// TwinCAT 3 PLC project p1
// ProgramVersion: 3.1.4023.0
// libraries:
//   Tc2_ControllerToolbox, * (Beckhoff Automation GmbH)
//   Tc2_EtherCAT, * (Beckhoff Automation GmbH)
//   Tc2_MC2, * (Beckhoff Automation GmbH)
//   Tc2_Standard, * (Beckhoff Automation GmbH)
//   Tc2_System, * (Beckhoff Automation GmbH)
//   Tc2_Utilities, * (Beckhoff Automation GmbH)
//   Tc3_Module, * (Beckhoff Automation GmbH)
// project tree:
//   DUTs/UR_10 _O2T_Registers/ UR_10_O2T_Registers.TcDUT, UR_O2T_bits_2.TcDUT, UR_O2T_floats_2.TcDUT, UR_O2T_int_2.TcDUT
//   DUTs/UR_3_T2O_Joints/ UR_3_T2O_Joints.TcDUT
//   DUTs/UR_4_T2O_TCP/ UR_4_T2O_TCP.TcDUT
//   DUTs/UR_5_T2O_BitRegisters/ UR_5_T2O_BitRegisters.TcDUT
//   DUTs/UR_6_T2O_IntRegisters/ UR_6_T2O_IntRegisters.TcDUT
//   DUTs/UR_7_T2O_FloatRegisters/ UR_7_T2O_FloatRegisters.TcDUT
//   DUTs/UR_9_O2T_Registers/ UR_9_O2T_Registers.TcDUT, UR_O2T_bits.TcDUT, UR_O2T_floats.TcDUT, UR_O2T_int.TcDUT
//   DUTs/Vision Struct/ ck_real_flag_data.TcDUT, Vision_data.TcDUT, Vision_flags.TcDUT, Vision_int_state.TcDUT
//   GVLs/MainProg Params/Constans/ VFUNCTION.TcGVL, _FUNCTION.TcGVL
//   GVLs/MainProg Params/Variables/ GLV_USER_FUN.TcGVL
//   GVLs/miscellaneus/ data_to_robot.TcGVL, Global_actual_velocity.TcGVL
//   GVLs/QRob/ QrCts.TcGVL
//   GVLs/QRob/Variables/ Global_Servo.TcGVL, QrRetVarState.TcGVL
//   GVLs/Robot Params/Constans/ RCts.TcGVL
//   GVLs/Robot Params/Variables/ Robot_UR5.TcGVL, Robot_UR3.TcGVL, UR3RetVarState.TcGVL, UR5RetVarState.TcGVL (not stored)
//   GVLs/Vision Params/Constants/ VCts.TcGVL
//   GVLs/Vision Params/Structs/ Vision_struct.TcGVL
//   GVLs/Vision Params/Variables/ VisionRetVarState.TcGVL
//   / PlcTask.TcTTO
//   POUs/POUs/Fuzzy/ Subsystem.TcPOU, trimf.TcPOU, trimf_l.TcPOU
//   POUs/POUs/IR_take_img/ get_images.TcPOU
//   POUs/POUs/l/ Atornillar_ur5.TcPOU, data_robot_ur5.TcPOU, data_robot_ur3.TcPOU, flip_byte_int.TcPOU, flip_real.TcPOU, flip_byte.TcPOU, flip_int.TcPOU, pulse_.TcPOU, limit_current.TcPOU
//   POUs/POUs/ MASTER_CTR.TcPOU
//   POUs/POUs/miscellaneous/ POU.TcPOU, profinet_UR3.TcPOU, profinet_UR5.TcPOU, UR3_Robot.TcPOU, UR5_robot.TcPOU
//   POUs/POUs/Qrob/QRob_functions/ Get_QRob_Pos.TcPOU, Temperature_Ctr.TcPOU, Qrob_control.TcPOU
//   POUs/POUs/Qrob/Qrob_State_Machine/ QRob_StateMachine.TcPOU
//   POUs/POUs/ROBOTS/Robot_functions/ ck_state.TcPOU, read_bool_flag.TcPOU, read_bool_flag_move.TcPOU, write_bool_flag.TcPOU, wr_GL_STATE.TcPOU (not stored), wr_state.TcPOU
//   POUs/POUs/ROBOTS/Robot_machine_state/ UR3_StateMachine.TcPOU, UR5_StateMachine.TcPOU
//   POUs/POUs/VISION/Vision_functions/ ck_state_v.TcPOU, ck_real_value.TcPOU, wr_real_value.TcPOU, wr_state_v.TcPOU
//   POUs/POUs/VISION/Vision_machines_states/ Vision_StateMachine.TcPOU
// real-time tasks:
//   TASK PlcTask2: cycle T#1ms, priority 4, ADS port 352
// motion (NC):
//   TASK NC-Task 1 SAF: cycle T#2ms, priority 6, ADS port 501
//   TASK NC-Task 1 SVB: cycle T#10ms, priority 10, ADS port 511
//   AXIS Axis 1 (id 1)
//     General: UnitName=°
//     Dynamic: Acceleration=321.75, Deceleration=321.75, Jerk=1070.01, FastAxisStopSignalType=3
//     Velo: RefSearch=70, RefSync=120, Fast=200, Maximum=225
//     PositionAreaControl: Enable=false
//     TargetPosControl: Enable=false
//     OtherSettings: AllowMotionCmdToSlave=true, DataPersistence=true
//     encoder EncType=19
//       EncPara: ScaleFactorNumerator=0.000686648, MaxCount=#xffffffff, ReferenceSystem=4
//         Inc: RefSyncInverse=false
//     drive DrvType=16
//       DrvPara: MaxCount=#xffffffff, DriveControlDWord=#x00020000
//         Analog: VeloReferenz=225, TorqueSetpointScale=1, ScaleFactorActTorque=1
//         TimeComp: TaskDelayCycles=1
//     controller CtrType=1
//       CtrPara: PriorControlFactor=1
//         PosDiffControl: Enable=false
//         Observer: BandWidth=20
// I/O:
//   DEVICE Device 5 (EtherCAT), AmsNetId 172.18.236.0.6.1
//     Drive 1 (ZeroErr Driver) [ZeroErr Driver]
//   DEVICE Device 7 (EtherCAT), AmsNetId 172.18.236.0.8.1
//     Term 4 (EK1100) [EK1100 EtherCAT Coupler (2A E-Bus)]
//       Term 5 (EL2809) [EL2809 16Ch. Dig. Output 24V, 0.5A]
//       Term 12 (EL1809) [EL1809 16Ch. Dig. Input 24V, 3ms]
//       Term 6 (EL6001) [EL6001 Interface (RS232)]
//       Term 4 (EL6631) [EL6631 PROFINET IO Controller]
//       Term 5 (EL6751) [EL6751 CANopen Master]
//       Term 6 (EL9011) [EL9011 End Terminal]
//   DEVICE Device 4 (EL6631), AmsNetId 172.18.236.0.5.1
//     uriodev1ur5 [Universal Robots A/S UR IO device, for PNIO controller with PDev 00000]
//       modules: Term 1 (DAP Module), Term 3 (1_T2O State), Term 4 (2_T2O IO), Term 5 (3_T2O Joints), Term 6 (4_T2O TCP), Term 7 (5_T2O General Purpose Bit Registers), Term 8 (6_T2O General Purpose Int Registers), Term 9 (7_T2O General Purpose Float Registers), Term 10 (8_O2T Robot IO), Term 11 (9_O2T General Purpose Registers 1), Term 12 (10_O2T General Purpose Registers 2)
//     uriodev1ur3 [Universal Robots A/S UR IO device, for PNIO controller with PDev 00000]
//       modules: Term 2 (DAP Module), Term 13 (1_T2O State), Term 14 (2_T2O IO), Term 15 (3_T2O Joints), Term 16 (4_T2O TCP), Term 17 (5_T2O General Purpose Bit Registers), Term 18 (6_T2O General Purpose Int Registers), Term 19 (7_T2O General Purpose Float Registers), Term 20 (8_O2T Robot IO), Term 21 (9_O2T General Purpose Registers 1), Term 22 (10_O2T General Purpose Registers 2)
// variable links:
//   NC-Task 1 SAF/Axes/Axis 1 <-> Device 5 (EtherCAT)/Drive 1 (ZeroErr Driver)
//     Drive/Inputs/In/nDataIn3[0] <-> Transmit PDO mapping 0/Torque Actual Value
//     Drive/Inputs/In/nDcOutputTime <-> InfoData/DcOutputShift
//     Drive/Inputs/In/nState1 <-> Transmit PDO mapping 0/Status word
//     Drive/Inputs/In/nState2 <-> Transmit PDO mapping 0/Status word @bit 8
//     Drive/Inputs/In/nState4 @bit 1 <-> WcState/InputToggle
//     Drive/Inputs/In/nState4 <-> WcState/WcState
//     Drive/Inputs/In/nState5 <-> Transmit PDO mapping 0/Modes of operation display
//     Drive/Outputs/Out/nCtrl1 <-> Receive PDO mapping 0/Control word
//     Drive/Outputs/Out/nCtrl2 <-> Receive PDO mapping 0/Control word @bit 8
//     Drive/Outputs/Out/nCtrl5 <-> Receive PDO mapping 0/Modes of operation
//     Drive/Outputs/Out/nDataOut1 <-> Receive PDO mapping 0/Target Position
//     Drive/Outputs/Out/nDataOut3[0] <-> Receive PDO mapping 0/Torque Offset
//     Drive/Outputs/Out/nDataOut4[0] <-> Receive PDO mapping 0/Target Torque
//     Enc/Inputs/In/nDataIn1 <-> Transmit PDO mapping 0/Position actual value
//     Enc/Inputs/In/nDataIn7 <-> Transmit PDO mapping 0/Actual velocity
//     Enc/Inputs/In/nDcInputTime <-> InfoData/DcInputShift
//     Enc/Inputs/In/nState4 @bit 1 <-> WcState/InputToggle
//     Enc/Inputs/In/nState4 <-> WcState/WcState
//   p1/p1 Instance <-> Device 4 (EL6631)/uriodev1ur3
//     PlcTask Inputs/Robot_UR3.UR_TCP/FLOAT14[0] <-> API/Term 16 (4_T2O TCP)/Subterm 20 (4_T2O TCP)/Inputs/T2O TCP[56]
//     PlcTask Inputs/Robot_UR3.UR_TCP/FLOAT14[1] <-> API/Term 16 (4_T2O TCP)/Subterm 20 (4_T2O TCP)/Inputs/T2O TCP[57]
//     PlcTask Inputs/Robot_UR3.UR_TCP/FLOAT14[2] <-> API/Term 16 (4_T2O TCP)/Subterm 20 (4_T2O TCP)/Inputs/T2O TCP[58]
//     PlcTask Inputs/Robot_UR3.UR_TCP/FLOAT14[3] <-> API/Term 16 (4_T2O TCP)/Subterm 20 (4_T2O TCP)/Inputs/T2O TCP[59]
//     PlcTask Inputs/Robot_UR3.UR_TCP/FLOAT15[0] <-> API/Term 16 (4_T2O TCP)/Subterm 20 (4_T2O TCP)/Inputs/T2O TCP[60]
//     PlcTask Inputs/Robot_UR3.UR_TCP/FLOAT15[1] <-> API/Term 16 (4_T2O TCP)/Subterm 20 (4_T2O TCP)/Inputs/T2O TCP[61]
//     PlcTask Inputs/Robot_UR3.UR_TCP/FLOAT15[2] <-> API/Term 16 (4_T2O TCP)/Subterm 20 (4_T2O TCP)/Inputs/T2O TCP[62]
//     PlcTask Inputs/Robot_UR3.UR_TCP/FLOAT15[3] <-> API/Term 16 (4_T2O TCP)/Subterm 20 (4_T2O TCP)/Inputs/T2O TCP[63]
//     PlcTask Inputs/Robot_UR3.UR_TCP/FLOAT16[0] <-> API/Term 16 (4_T2O TCP)/Subterm 20 (4_T2O TCP)/Inputs/T2O TCP[64]
//     PlcTask Inputs/Robot_UR3.UR_TCP/FLOAT16[1] <-> API/Term 16 (4_T2O TCP)/Subterm 20 (4_T2O TCP)/Inputs/T2O TCP[65]
//     PlcTask Inputs/Robot_UR3.UR_TCP/FLOAT16[2] <-> API/Term 16 (4_T2O TCP)/Subterm 20 (4_T2O TCP)/Inputs/T2O TCP[66]
//     PlcTask Inputs/Robot_UR3.UR_TCP/FLOAT16[3] <-> API/Term 16 (4_T2O TCP)/Subterm 20 (4_T2O TCP)/Inputs/T2O TCP[67]
//     PlcTask Inputs/Robot_UR3.UR_TCP/FLOAT17[0] <-> API/Term 16 (4_T2O TCP)/Subterm 20 (4_T2O TCP)/Inputs/T2O TCP[68]
//     PlcTask Inputs/Robot_UR3.UR_TCP/FLOAT17[1] <-> API/Term 16 (4_T2O TCP)/Subterm 20 (4_T2O TCP)/Inputs/T2O TCP[69]
//     PlcTask Inputs/Robot_UR3.UR_TCP/FLOAT17[2] <-> API/Term 16 (4_T2O TCP)/Subterm 20 (4_T2O TCP)/Inputs/T2O TCP[70]
//     PlcTask Inputs/Robot_UR3.UR_TCP/FLOAT17[3] <-> API/Term 16 (4_T2O TCP)/Subterm 20 (4_T2O TCP)/Inputs/T2O TCP[71]
//     PlcTask Inputs/Robot_UR3.UR_TCP/FLOAT18[0] <-> API/Term 16 (4_T2O TCP)/Subterm 20 (4_T2O TCP)/Inputs/T2O TCP[72]
//     PlcTask Inputs/Robot_UR3.UR_TCP/FLOAT18[1] <-> API/Term 16 (4_T2O TCP)/Subterm 20 (4_T2O TCP)/Inputs/T2O TCP[73]
//     PlcTask Inputs/Robot_UR3.UR_TCP/FLOAT18[2] <-> API/Term 16 (4_T2O TCP)/Subterm 20 (4_T2O TCP)/Inputs/T2O TCP[74]
//     PlcTask Inputs/Robot_UR3.UR_TCP/FLOAT18[3] <-> API/Term 16 (4_T2O TCP)/Subterm 20 (4_T2O TCP)/Inputs/T2O TCP[75]
//     PlcTask Inputs/Robot_UR3.UR_outputs/B{0..56 step 8} <-> API/Term 17 (5_T2O General Purpose Bit Registers)/Subterm 21 (5_T2O General Purpose Bit Registers)/Inputs/T2O Bit Registers[{0..7}]  (8 links)
//     PlcTask Inputs/Robot_UR3.UR_outputs/B1 <-> API/Term 17 (5_T2O General Purpose Bit Registers)/Subterm 21 (5_T2O General Purpose Bit Registers)/Inputs/T2O Bit Registers[0] @bit 1
//     PlcTask Inputs/Robot_UR3.UR_outputs/B10 <-> API/Term 17 (5_T2O General Purpose Bit Registers)/Subterm 21 (5_T2O General Purpose Bit Registers)/Inputs/T2O Bit Registers[1] @bit 2
//     PlcTask Inputs/Robot_UR3.UR_outputs/B11 <-> API/Term 17 (5_T2O General Purpose Bit Registers)/Subterm 21 (5_T2O General Purpose Bit Registers)/Inputs/T2O Bit Registers[1] @bit 3
//     PlcTask Inputs/Robot_UR3.UR_outputs/B12 <-> API/Term 17 (5_T2O General Purpose Bit Registers)/Subterm 21 (5_T2O General Purpose Bit Registers)/Inputs/T2O Bit Registers[1] @bit 4
//     PlcTask Inputs/Robot_UR3.UR_outputs/B13 <-> API/Term 17 (5_T2O General Purpose Bit Registers)/Subterm 21 (5_T2O General Purpose Bit Registers)/Inputs/T2O Bit Registers[1] @bit 5
//     PlcTask Inputs/Robot_UR3.UR_outputs/B14 <-> API/Term 17 (5_T2O General Purpose Bit Registers)/Subterm 21 (5_T2O General Purpose Bit Registers)/Inputs/T2O Bit Registers[1] @bit 6
//     PlcTask Inputs/Robot_UR3.UR_outputs/B15 <-> API/Term 17 (5_T2O General Purpose Bit Registers)/Subterm 21 (5_T2O General Purpose Bit Registers)/Inputs/T2O Bit Registers[1] @bit 7
//     PlcTask Inputs/Robot_UR3.UR_outputs/B17 <-> API/Term 17 (5_T2O General Purpose Bit Registers)/Subterm 21 (5_T2O General Purpose Bit Registers)/Inputs/T2O Bit Registers[2] @bit 1
//     PlcTask Inputs/Robot_UR3.UR_outputs/B18 <-> API/Term 17 (5_T2O General Purpose Bit Registers)/Subterm 21 (5_T2O General Purpose Bit Registers)/Inputs/T2O Bit Registers[2] @bit 2
//     PlcTask Inputs/Robot_UR3.UR_outputs/B19 <-> API/Term 17 (5_T2O General Purpose Bit Registers)/Subterm 21 (5_T2O General Purpose Bit Registers)/Inputs/T2O Bit Registers[2] @bit 3
//     PlcTask Inputs/Robot_UR3.UR_outputs/B2 <-> API/Term 17 (5_T2O General Purpose Bit Registers)/Subterm 21 (5_T2O General Purpose Bit Registers)/Inputs/T2O Bit Registers[0] @bit 2
//     PlcTask Inputs/Robot_UR3.UR_outputs/B20 <-> API/Term 17 (5_T2O General Purpose Bit Registers)/Subterm 21 (5_T2O General Purpose Bit Registers)/Inputs/T2O Bit Registers[2] @bit 4
//     PlcTask Inputs/Robot_UR3.UR_outputs/B21 <-> API/Term 17 (5_T2O General Purpose Bit Registers)/Subterm 21 (5_T2O General Purpose Bit Registers)/Inputs/T2O Bit Registers[2] @bit 5
//     PlcTask Inputs/Robot_UR3.UR_outputs/B22 <-> API/Term 17 (5_T2O General Purpose Bit Registers)/Subterm 21 (5_T2O General Purpose Bit Registers)/Inputs/T2O Bit Registers[2] @bit 6
//     PlcTask Inputs/Robot_UR3.UR_outputs/B23 <-> API/Term 17 (5_T2O General Purpose Bit Registers)/Subterm 21 (5_T2O General Purpose Bit Registers)/Inputs/T2O Bit Registers[2] @bit 7
//     PlcTask Inputs/Robot_UR3.UR_outputs/B25 <-> API/Term 17 (5_T2O General Purpose Bit Registers)/Subterm 21 (5_T2O General Purpose Bit Registers)/Inputs/T2O Bit Registers[3] @bit 1
//     PlcTask Inputs/Robot_UR3.UR_outputs/B26 <-> API/Term 17 (5_T2O General Purpose Bit Registers)/Subterm 21 (5_T2O General Purpose Bit Registers)/Inputs/T2O Bit Registers[3] @bit 2
//     PlcTask Inputs/Robot_UR3.UR_outputs/B27 <-> API/Term 17 (5_T2O General Purpose Bit Registers)/Subterm 21 (5_T2O General Purpose Bit Registers)/Inputs/T2O Bit Registers[3] @bit 3
//     PlcTask Inputs/Robot_UR3.UR_outputs/B28 <-> API/Term 17 (5_T2O General Purpose Bit Registers)/Subterm 21 (5_T2O General Purpose Bit Registers)/Inputs/T2O Bit Registers[3] @bit 4
//     PlcTask Inputs/Robot_UR3.UR_outputs/B29 <-> API/Term 17 (5_T2O General Purpose Bit Registers)/Subterm 21 (5_T2O General Purpose Bit Registers)/Inputs/T2O Bit Registers[3] @bit 5
//     PlcTask Inputs/Robot_UR3.UR_outputs/B3 <-> API/Term 17 (5_T2O General Purpose Bit Registers)/Subterm 21 (5_T2O General Purpose Bit Registers)/Inputs/T2O Bit Registers[0] @bit 3
//     PlcTask Inputs/Robot_UR3.UR_outputs/B30 <-> API/Term 17 (5_T2O General Purpose Bit Registers)/Subterm 21 (5_T2O General Purpose Bit Registers)/Inputs/T2O Bit Registers[3] @bit 6
//     PlcTask Inputs/Robot_UR3.UR_outputs/B31 <-> API/Term 17 (5_T2O General Purpose Bit Registers)/Subterm 21 (5_T2O General Purpose Bit Registers)/Inputs/T2O Bit Registers[3] @bit 7
//     PlcTask Inputs/Robot_UR3.UR_outputs/B33 <-> API/Term 17 (5_T2O General Purpose Bit Registers)/Subterm 21 (5_T2O General Purpose Bit Registers)/Inputs/T2O Bit Registers[4] @bit 1
//     PlcTask Inputs/Robot_UR3.UR_outputs/B34 <-> API/Term 17 (5_T2O General Purpose Bit Registers)/Subterm 21 (5_T2O General Purpose Bit Registers)/Inputs/T2O Bit Registers[4] @bit 2
//     PlcTask Inputs/Robot_UR3.UR_outputs/B35 <-> API/Term 17 (5_T2O General Purpose Bit Registers)/Subterm 21 (5_T2O General Purpose Bit Registers)/Inputs/T2O Bit Registers[4] @bit 3
//     PlcTask Inputs/Robot_UR3.UR_outputs/B36 <-> API/Term 17 (5_T2O General Purpose Bit Registers)/Subterm 21 (5_T2O General Purpose Bit Registers)/Inputs/T2O Bit Registers[4] @bit 4
//     PlcTask Inputs/Robot_UR3.UR_outputs/B37 <-> API/Term 17 (5_T2O General Purpose Bit Registers)/Subterm 21 (5_T2O General Purpose Bit Registers)/Inputs/T2O Bit Registers[4] @bit 5
//     PlcTask Inputs/Robot_UR3.UR_outputs/B38 <-> API/Term 17 (5_T2O General Purpose Bit Registers)/Subterm 21 (5_T2O General Purpose Bit Registers)/Inputs/T2O Bit Registers[4] @bit 6
//     PlcTask Inputs/Robot_UR3.UR_outputs/B39 <-> API/Term 17 (5_T2O General Purpose Bit Registers)/Subterm 21 (5_T2O General Purpose Bit Registers)/Inputs/T2O Bit Registers[4] @bit 7
//     PlcTask Inputs/Robot_UR3.UR_outputs/B4 <-> API/Term 17 (5_T2O General Purpose Bit Registers)/Subterm 21 (5_T2O General Purpose Bit Registers)/Inputs/T2O Bit Registers[0] @bit 4
//     PlcTask Inputs/Robot_UR3.UR_outputs/B41 <-> API/Term 17 (5_T2O General Purpose Bit Registers)/Subterm 21 (5_T2O General Purpose Bit Registers)/Inputs/T2O Bit Registers[5] @bit 1
//     PlcTask Inputs/Robot_UR3.UR_outputs/B42 <-> API/Term 17 (5_T2O General Purpose Bit Registers)/Subterm 21 (5_T2O General Purpose Bit Registers)/Inputs/T2O Bit Registers[5] @bit 2
//     PlcTask Inputs/Robot_UR3.UR_outputs/B43 <-> API/Term 17 (5_T2O General Purpose Bit Registers)/Subterm 21 (5_T2O General Purpose Bit Registers)/Inputs/T2O Bit Registers[5] @bit 3
//     PlcTask Inputs/Robot_UR3.UR_outputs/B44 <-> API/Term 17 (5_T2O General Purpose Bit Registers)/Subterm 21 (5_T2O General Purpose Bit Registers)/Inputs/T2O Bit Registers[5] @bit 4
//     PlcTask Inputs/Robot_UR3.UR_outputs/B45 <-> API/Term 17 (5_T2O General Purpose Bit Registers)/Subterm 21 (5_T2O General Purpose Bit Registers)/Inputs/T2O Bit Registers[5] @bit 5
//     PlcTask Inputs/Robot_UR3.UR_outputs/B46 <-> API/Term 17 (5_T2O General Purpose Bit Registers)/Subterm 21 (5_T2O General Purpose Bit Registers)/Inputs/T2O Bit Registers[5] @bit 6
//     PlcTask Inputs/Robot_UR3.UR_outputs/B47 <-> API/Term 17 (5_T2O General Purpose Bit Registers)/Subterm 21 (5_T2O General Purpose Bit Registers)/Inputs/T2O Bit Registers[5] @bit 7
//     PlcTask Inputs/Robot_UR3.UR_outputs/B49 <-> API/Term 17 (5_T2O General Purpose Bit Registers)/Subterm 21 (5_T2O General Purpose Bit Registers)/Inputs/T2O Bit Registers[6] @bit 1
//     PlcTask Inputs/Robot_UR3.UR_outputs/B5 <-> API/Term 17 (5_T2O General Purpose Bit Registers)/Subterm 21 (5_T2O General Purpose Bit Registers)/Inputs/T2O Bit Registers[0] @bit 5
//     PlcTask Inputs/Robot_UR3.UR_outputs/B50 <-> API/Term 17 (5_T2O General Purpose Bit Registers)/Subterm 21 (5_T2O General Purpose Bit Registers)/Inputs/T2O Bit Registers[6] @bit 2
//     PlcTask Inputs/Robot_UR3.UR_outputs/B51 <-> API/Term 17 (5_T2O General Purpose Bit Registers)/Subterm 21 (5_T2O General Purpose Bit Registers)/Inputs/T2O Bit Registers[6] @bit 3
//     PlcTask Inputs/Robot_UR3.UR_outputs/B52 <-> API/Term 17 (5_T2O General Purpose Bit Registers)/Subterm 21 (5_T2O General Purpose Bit Registers)/Inputs/T2O Bit Registers[6] @bit 4
//     PlcTask Inputs/Robot_UR3.UR_outputs/B53 <-> API/Term 17 (5_T2O General Purpose Bit Registers)/Subterm 21 (5_T2O General Purpose Bit Registers)/Inputs/T2O Bit Registers[6] @bit 5
//     PlcTask Inputs/Robot_UR3.UR_outputs/B54 <-> API/Term 17 (5_T2O General Purpose Bit Registers)/Subterm 21 (5_T2O General Purpose Bit Registers)/Inputs/T2O Bit Registers[6] @bit 6
//     PlcTask Inputs/Robot_UR3.UR_outputs/B55 <-> API/Term 17 (5_T2O General Purpose Bit Registers)/Subterm 21 (5_T2O General Purpose Bit Registers)/Inputs/T2O Bit Registers[6] @bit 7
//     PlcTask Inputs/Robot_UR3.UR_outputs/B57 <-> API/Term 17 (5_T2O General Purpose Bit Registers)/Subterm 21 (5_T2O General Purpose Bit Registers)/Inputs/T2O Bit Registers[7] @bit 1
//     PlcTask Inputs/Robot_UR3.UR_outputs/B58 <-> API/Term 17 (5_T2O General Purpose Bit Registers)/Subterm 21 (5_T2O General Purpose Bit Registers)/Inputs/T2O Bit Registers[7] @bit 2
//     PlcTask Inputs/Robot_UR3.UR_outputs/B59 <-> API/Term 17 (5_T2O General Purpose Bit Registers)/Subterm 21 (5_T2O General Purpose Bit Registers)/Inputs/T2O Bit Registers[7] @bit 3
//     PlcTask Inputs/Robot_UR3.UR_outputs/B6 <-> API/Term 17 (5_T2O General Purpose Bit Registers)/Subterm 21 (5_T2O General Purpose Bit Registers)/Inputs/T2O Bit Registers[0] @bit 6
//     PlcTask Inputs/Robot_UR3.UR_outputs/B60 <-> API/Term 17 (5_T2O General Purpose Bit Registers)/Subterm 21 (5_T2O General Purpose Bit Registers)/Inputs/T2O Bit Registers[7] @bit 4
//     PlcTask Inputs/Robot_UR3.UR_outputs/B61 <-> API/Term 17 (5_T2O General Purpose Bit Registers)/Subterm 21 (5_T2O General Purpose Bit Registers)/Inputs/T2O Bit Registers[7] @bit 5
//     PlcTask Inputs/Robot_UR3.UR_outputs/B62 <-> API/Term 17 (5_T2O General Purpose Bit Registers)/Subterm 21 (5_T2O General Purpose Bit Registers)/Inputs/T2O Bit Registers[7] @bit 6
//     PlcTask Inputs/Robot_UR3.UR_outputs/B63 <-> API/Term 17 (5_T2O General Purpose Bit Registers)/Subterm 21 (5_T2O General Purpose Bit Registers)/Inputs/T2O Bit Registers[7] @bit 7
//     PlcTask Inputs/Robot_UR3.UR_outputs/B7 <-> API/Term 17 (5_T2O General Purpose Bit Registers)/Subterm 21 (5_T2O General Purpose Bit Registers)/Inputs/T2O Bit Registers[0] @bit 7
//     PlcTask Inputs/Robot_UR3.UR_outputs/B9 <-> API/Term 17 (5_T2O General Purpose Bit Registers)/Subterm 21 (5_T2O General Purpose Bit Registers)/Inputs/T2O Bit Registers[1] @bit 1
//     PlcTask Inputs/Robot_UR3.UR_outputs_int/INT0[0] <-> API/Term 18 (6_T2O General Purpose Int Registers)/Subterm 22 (6_T2O General Purpose Int Registers)/Inputs/T2O Int Registers[0]
//     PlcTask Inputs/Robot_UR3.UR_outputs_int/INT0[1] <-> API/Term 18 (6_T2O General Purpose Int Registers)/Subterm 22 (6_T2O General Purpose Int Registers)/Inputs/T2O Int Registers[1]
//     PlcTask Inputs/Robot_UR3.UR_outputs_int/INT0[2] <-> API/Term 18 (6_T2O General Purpose Int Registers)/Subterm 22 (6_T2O General Purpose Int Registers)/Inputs/T2O Int Registers[2]
//     PlcTask Inputs/Robot_UR3.UR_outputs_int/INT0[3] <-> API/Term 18 (6_T2O General Purpose Int Registers)/Subterm 22 (6_T2O General Purpose Int Registers)/Inputs/T2O Int Registers[3]
//     PlcTask Inputs/Robot_UR3.UR_outputs_int/INT1[0] <-> API/Term 18 (6_T2O General Purpose Int Registers)/Subterm 22 (6_T2O General Purpose Int Registers)/Inputs/T2O Int Registers[4]
//     PlcTask Inputs/Robot_UR3.UR_outputs_int/INT1[1] <-> API/Term 18 (6_T2O General Purpose Int Registers)/Subterm 22 (6_T2O General Purpose Int Registers)/Inputs/T2O Int Registers[5]
//     PlcTask Inputs/Robot_UR3.UR_outputs_int/INT1[2] <-> API/Term 18 (6_T2O General Purpose Int Registers)/Subterm 22 (6_T2O General Purpose Int Registers)/Inputs/T2O Int Registers[6]
//     PlcTask Inputs/Robot_UR3.UR_outputs_int/INT1[3] <-> API/Term 18 (6_T2O General Purpose Int Registers)/Subterm 22 (6_T2O General Purpose Int Registers)/Inputs/T2O Int Registers[7]
//     PlcTask Inputs/Robot_UR3.UR_outputs_int/INT2[0] <-> API/Term 18 (6_T2O General Purpose Int Registers)/Subterm 22 (6_T2O General Purpose Int Registers)/Inputs/T2O Int Registers[8]
//     PlcTask Inputs/Robot_UR3.UR_outputs_int/INT2[1] <-> API/Term 18 (6_T2O General Purpose Int Registers)/Subterm 22 (6_T2O General Purpose Int Registers)/Inputs/T2O Int Registers[9]
//     PlcTask Inputs/Robot_UR3.UR_outputs_int/INT2[2] <-> API/Term 18 (6_T2O General Purpose Int Registers)/Subterm 22 (6_T2O General Purpose Int Registers)/Inputs/T2O Int Registers[10]
//     PlcTask Inputs/Robot_UR3.UR_outputs_int/INT2[3] <-> API/Term 18 (6_T2O General Purpose Int Registers)/Subterm 22 (6_T2O General Purpose Int Registers)/Inputs/T2O Int Registers[11]
//     PlcTask Inputs/Robot_UR3.UR_outputs_int/INT3[0] <-> API/Term 18 (6_T2O General Purpose Int Registers)/Subterm 22 (6_T2O General Purpose Int Registers)/Inputs/T2O Int Registers[12]
//     PlcTask Inputs/Robot_UR3.UR_outputs_int/INT3[1] <-> API/Term 18 (6_T2O General Purpose Int Registers)/Subterm 22 (6_T2O General Purpose Int Registers)/Inputs/T2O Int Registers[13]
//     PlcTask Inputs/Robot_UR3.UR_outputs_int/INT3[2] <-> API/Term 18 (6_T2O General Purpose Int Registers)/Subterm 22 (6_T2O General Purpose Int Registers)/Inputs/T2O Int Registers[14]
//     PlcTask Inputs/Robot_UR3.UR_outputs_int/INT3[3] <-> API/Term 18 (6_T2O General Purpose Int Registers)/Subterm 22 (6_T2O General Purpose Int Registers)/Inputs/T2O Int Registers[15]
//     PlcTask Inputs/Robot_UR3.UR_outputs_int/INT4[0] <-> API/Term 18 (6_T2O General Purpose Int Registers)/Subterm 22 (6_T2O General Purpose Int Registers)/Inputs/T2O Int Registers[16]
//     PlcTask Inputs/Robot_UR3.UR_outputs_int/INT4[1] <-> API/Term 18 (6_T2O General Purpose Int Registers)/Subterm 22 (6_T2O General Purpose Int Registers)/Inputs/T2O Int Registers[17]
//     PlcTask Inputs/Robot_UR3.UR_outputs_int/INT4[2] <-> API/Term 18 (6_T2O General Purpose Int Registers)/Subterm 22 (6_T2O General Purpose Int Registers)/Inputs/T2O Int Registers[18]
//     PlcTask Inputs/Robot_UR3.UR_outputs_int/INT4[3] <-> API/Term 18 (6_T2O General Purpose Int Registers)/Subterm 22 (6_T2O General Purpose Int Registers)/Inputs/T2O Int Registers[19]
//     PlcTask Inputs/Robot_UR3.UR_outputs_int/INT5[0] <-> API/Term 18 (6_T2O General Purpose Int Registers)/Subterm 22 (6_T2O General Purpose Int Registers)/Inputs/T2O Int Registers[20]
//     PlcTask Inputs/Robot_UR3.UR_outputs_int/INT5[1] <-> API/Term 18 (6_T2O General Purpose Int Registers)/Subterm 22 (6_T2O General Purpose Int Registers)/Inputs/T2O Int Registers[21]
//     PlcTask Inputs/Robot_UR3.UR_outputs_int/INT5[2] <-> API/Term 18 (6_T2O General Purpose Int Registers)/Subterm 22 (6_T2O General Purpose Int Registers)/Inputs/T2O Int Registers[22]
//     PlcTask Inputs/Robot_UR3.UR_outputs_int/INT5[3] <-> API/Term 18 (6_T2O General Purpose Int Registers)/Subterm 22 (6_T2O General Purpose Int Registers)/Inputs/T2O Int Registers[23]
//     PlcTask Inputs/Robot_UR3.UR_outputs_int/INT6[0] <-> API/Term 18 (6_T2O General Purpose Int Registers)/Subterm 22 (6_T2O General Purpose Int Registers)/Inputs/T2O Int Registers[24]
//     PlcTask Inputs/Robot_UR3.UR_outputs_int/INT6[1] <-> API/Term 18 (6_T2O General Purpose Int Registers)/Subterm 22 (6_T2O General Purpose Int Registers)/Inputs/T2O Int Registers[25]
//     PlcTask Inputs/Robot_UR3.UR_outputs_int/INT6[2] <-> API/Term 18 (6_T2O General Purpose Int Registers)/Subterm 22 (6_T2O General Purpose Int Registers)/Inputs/T2O Int Registers[26]
//     PlcTask Inputs/Robot_UR3.UR_outputs_int/INT6[3] <-> API/Term 18 (6_T2O General Purpose Int Registers)/Subterm 22 (6_T2O General Purpose Int Registers)/Inputs/T2O Int Registers[27]
//     PlcTask Outputs/Robot_UR3.UR_inputs/Bits/B{0..24 step 8} <-> API/Term 21 (9_O2T General Purpose Registers 1)/Subterm 25 (9_O2T General Purpose Registers 1)/Outputs/O2T Reg 1[{0..3}]  (4 links)
//     PlcTask Outputs/Robot_UR3.UR_inputs/Bits/B1 <-> API/Term 21 (9_O2T General Purpose Registers 1)/Subterm 25 (9_O2T General Purpose Registers 1)/Outputs/O2T Reg 1[0] @bit 1
//     PlcTask Outputs/Robot_UR3.UR_inputs/Bits/B10 <-> API/Term 21 (9_O2T General Purpose Registers 1)/Subterm 25 (9_O2T General Purpose Registers 1)/Outputs/O2T Reg 1[1] @bit 2
//     PlcTask Outputs/Robot_UR3.UR_inputs/Bits/B11 <-> API/Term 21 (9_O2T General Purpose Registers 1)/Subterm 25 (9_O2T General Purpose Registers 1)/Outputs/O2T Reg 1[1] @bit 3
//     PlcTask Outputs/Robot_UR3.UR_inputs/Bits/B12 <-> API/Term 21 (9_O2T General Purpose Registers 1)/Subterm 25 (9_O2T General Purpose Registers 1)/Outputs/O2T Reg 1[1] @bit 4
//     PlcTask Outputs/Robot_UR3.UR_inputs/Bits/B13 <-> API/Term 21 (9_O2T General Purpose Registers 1)/Subterm 25 (9_O2T General Purpose Registers 1)/Outputs/O2T Reg 1[1] @bit 5
//     PlcTask Outputs/Robot_UR3.UR_inputs/Bits/B14 <-> API/Term 21 (9_O2T General Purpose Registers 1)/Subterm 25 (9_O2T General Purpose Registers 1)/Outputs/O2T Reg 1[1] @bit 6
//     PlcTask Outputs/Robot_UR3.UR_inputs/Bits/B15 <-> API/Term 21 (9_O2T General Purpose Registers 1)/Subterm 25 (9_O2T General Purpose Registers 1)/Outputs/O2T Reg 1[1] @bit 7
//     PlcTask Outputs/Robot_UR3.UR_inputs/Bits/B17 <-> API/Term 21 (9_O2T General Purpose Registers 1)/Subterm 25 (9_O2T General Purpose Registers 1)/Outputs/O2T Reg 1[2] @bit 1
//     PlcTask Outputs/Robot_UR3.UR_inputs/Bits/B18 <-> API/Term 21 (9_O2T General Purpose Registers 1)/Subterm 25 (9_O2T General Purpose Registers 1)/Outputs/O2T Reg 1[2] @bit 2
//     PlcTask Outputs/Robot_UR3.UR_inputs/Bits/B19 <-> API/Term 21 (9_O2T General Purpose Registers 1)/Subterm 25 (9_O2T General Purpose Registers 1)/Outputs/O2T Reg 1[2] @bit 3
//     PlcTask Outputs/Robot_UR3.UR_inputs/Bits/B2 <-> API/Term 21 (9_O2T General Purpose Registers 1)/Subterm 25 (9_O2T General Purpose Registers 1)/Outputs/O2T Reg 1[0] @bit 2
//     PlcTask Outputs/Robot_UR3.UR_inputs/Bits/B20 <-> API/Term 21 (9_O2T General Purpose Registers 1)/Subterm 25 (9_O2T General Purpose Registers 1)/Outputs/O2T Reg 1[2] @bit 4
//     PlcTask Outputs/Robot_UR3.UR_inputs/Bits/B21 <-> API/Term 21 (9_O2T General Purpose Registers 1)/Subterm 25 (9_O2T General Purpose Registers 1)/Outputs/O2T Reg 1[2] @bit 5
//     PlcTask Outputs/Robot_UR3.UR_inputs/Bits/B22 <-> API/Term 21 (9_O2T General Purpose Registers 1)/Subterm 25 (9_O2T General Purpose Registers 1)/Outputs/O2T Reg 1[2] @bit 6
//     PlcTask Outputs/Robot_UR3.UR_inputs/Bits/B23 <-> API/Term 21 (9_O2T General Purpose Registers 1)/Subterm 25 (9_O2T General Purpose Registers 1)/Outputs/O2T Reg 1[2] @bit 7
//     PlcTask Outputs/Robot_UR3.UR_inputs/Bits/B25 <-> API/Term 21 (9_O2T General Purpose Registers 1)/Subterm 25 (9_O2T General Purpose Registers 1)/Outputs/O2T Reg 1[3] @bit 1
//     PlcTask Outputs/Robot_UR3.UR_inputs/Bits/B26 <-> API/Term 21 (9_O2T General Purpose Registers 1)/Subterm 25 (9_O2T General Purpose Registers 1)/Outputs/O2T Reg 1[3] @bit 2
//     PlcTask Outputs/Robot_UR3.UR_inputs/Bits/B27 <-> API/Term 21 (9_O2T General Purpose Registers 1)/Subterm 25 (9_O2T General Purpose Registers 1)/Outputs/O2T Reg 1[3] @bit 3
//     PlcTask Outputs/Robot_UR3.UR_inputs/Bits/B28 <-> API/Term 21 (9_O2T General Purpose Registers 1)/Subterm 25 (9_O2T General Purpose Registers 1)/Outputs/O2T Reg 1[3] @bit 4
//     PlcTask Outputs/Robot_UR3.UR_inputs/Bits/B29 <-> API/Term 21 (9_O2T General Purpose Registers 1)/Subterm 25 (9_O2T General Purpose Registers 1)/Outputs/O2T Reg 1[3] @bit 5
//     PlcTask Outputs/Robot_UR3.UR_inputs/Bits/B3 <-> API/Term 21 (9_O2T General Purpose Registers 1)/Subterm 25 (9_O2T General Purpose Registers 1)/Outputs/O2T Reg 1[0] @bit 3
//     PlcTask Outputs/Robot_UR3.UR_inputs/Bits/B30 <-> API/Term 21 (9_O2T General Purpose Registers 1)/Subterm 25 (9_O2T General Purpose Registers 1)/Outputs/O2T Reg 1[3] @bit 6
//     PlcTask Outputs/Robot_UR3.UR_inputs/Bits/B31 <-> API/Term 21 (9_O2T General Purpose Registers 1)/Subterm 25 (9_O2T General Purpose Registers 1)/Outputs/O2T Reg 1[3] @bit 7
//     PlcTask Outputs/Robot_UR3.UR_inputs/Bits/B4 <-> API/Term 21 (9_O2T General Purpose Registers 1)/Subterm 25 (9_O2T General Purpose Registers 1)/Outputs/O2T Reg 1[0] @bit 4
//     PlcTask Outputs/Robot_UR3.UR_inputs/Bits/B5 <-> API/Term 21 (9_O2T General Purpose Registers 1)/Subterm 25 (9_O2T General Purpose Registers 1)/Outputs/O2T Reg 1[0] @bit 5
//     PlcTask Outputs/Robot_UR3.UR_inputs/Bits/B6 <-> API/Term 21 (9_O2T General Purpose Registers 1)/Subterm 25 (9_O2T General Purpose Registers 1)/Outputs/O2T Reg 1[0] @bit 6
//     PlcTask Outputs/Robot_UR3.UR_inputs/Bits/B7 <-> API/Term 21 (9_O2T General Purpose Registers 1)/Subterm 25 (9_O2T General Purpose Registers 1)/Outputs/O2T Reg 1[0] @bit 7
//     PlcTask Outputs/Robot_UR3.UR_inputs/Bits/B9 <-> API/Term 21 (9_O2T General Purpose Registers 1)/Subterm 25 (9_O2T General Purpose Registers 1)/Outputs/O2T Reg 1[1] @bit 1
//     PlcTask Outputs/Robot_UR3.UR_inputs/Ints/INT0[0] <-> API/Term 21 (9_O2T General Purpose Registers 1)/Subterm 25 (9_O2T General Purpose Registers 1)/Outputs/O2T Reg 1[4]
//     PlcTask Outputs/Robot_UR3.UR_inputs/Ints/INT0[1] <-> API/Term 21 (9_O2T General Purpose Registers 1)/Subterm 25 (9_O2T General Purpose Registers 1)/Outputs/O2T Reg 1[5]
//     PlcTask Outputs/Robot_UR3.UR_inputs/Ints/INT0[2] <-> API/Term 21 (9_O2T General Purpose Registers 1)/Subterm 25 (9_O2T General Purpose Registers 1)/Outputs/O2T Reg 1[6]
//     PlcTask Outputs/Robot_UR3.UR_inputs/Ints/INT0[3] <-> API/Term 21 (9_O2T General Purpose Registers 1)/Subterm 25 (9_O2T General Purpose Registers 1)/Outputs/O2T Reg 1[7]
//     PlcTask Outputs/Robot_UR3.UR_inputs/Ints/INT10[0] <-> API/Term 21 (9_O2T General Purpose Registers 1)/Subterm 25 (9_O2T General Purpose Registers 1)/Outputs/O2T Reg 1[44]
//     PlcTask Outputs/Robot_UR3.UR_inputs/Ints/INT10[1] <-> API/Term 21 (9_O2T General Purpose Registers 1)/Subterm 25 (9_O2T General Purpose Registers 1)/Outputs/O2T Reg 1[45]
//     PlcTask Outputs/Robot_UR3.UR_inputs/Ints/INT10[2] <-> API/Term 21 (9_O2T General Purpose Registers 1)/Subterm 25 (9_O2T General Purpose Registers 1)/Outputs/O2T Reg 1[46]
//     PlcTask Outputs/Robot_UR3.UR_inputs/Ints/INT10[3] <-> API/Term 21 (9_O2T General Purpose Registers 1)/Subterm 25 (9_O2T General Purpose Registers 1)/Outputs/O2T Reg 1[47]
//     PlcTask Outputs/Robot_UR3.UR_inputs/Ints/INT11[0] <-> API/Term 21 (9_O2T General Purpose Registers 1)/Subterm 25 (9_O2T General Purpose Registers 1)/Outputs/O2T Reg 1[48]
//     PlcTask Outputs/Robot_UR3.UR_inputs/Ints/INT11[1] <-> API/Term 21 (9_O2T General Purpose Registers 1)/Subterm 25 (9_O2T General Purpose Registers 1)/Outputs/O2T Reg 1[49]
//     PlcTask Outputs/Robot_UR3.UR_inputs/Ints/INT11[2] <-> API/Term 21 (9_O2T General Purpose Registers 1)/Subterm 25 (9_O2T General Purpose Registers 1)/Outputs/O2T Reg 1[50]
//     PlcTask Outputs/Robot_UR3.UR_inputs/Ints/INT11[3] <-> API/Term 21 (9_O2T General Purpose Registers 1)/Subterm 25 (9_O2T General Purpose Registers 1)/Outputs/O2T Reg 1[51]
//     PlcTask Outputs/Robot_UR3.UR_inputs/Ints/INT1[0] <-> API/Term 21 (9_O2T General Purpose Registers 1)/Subterm 25 (9_O2T General Purpose Registers 1)/Outputs/O2T Reg 1[8]
//     PlcTask Outputs/Robot_UR3.UR_inputs/Ints/INT1[1] <-> API/Term 21 (9_O2T General Purpose Registers 1)/Subterm 25 (9_O2T General Purpose Registers 1)/Outputs/O2T Reg 1[9]
//     PlcTask Outputs/Robot_UR3.UR_inputs/Ints/INT1[2] <-> API/Term 21 (9_O2T General Purpose Registers 1)/Subterm 25 (9_O2T General Purpose Registers 1)/Outputs/O2T Reg 1[10]
//     PlcTask Outputs/Robot_UR3.UR_inputs/Ints/INT1[3] <-> API/Term 21 (9_O2T General Purpose Registers 1)/Subterm 25 (9_O2T General Purpose Registers 1)/Outputs/O2T Reg 1[11]
//     PlcTask Outputs/Robot_UR3.UR_inputs/Ints/INT2[0] <-> API/Term 21 (9_O2T General Purpose Registers 1)/Subterm 25 (9_O2T General Purpose Registers 1)/Outputs/O2T Reg 1[12]
//     PlcTask Outputs/Robot_UR3.UR_inputs/Ints/INT2[1] <-> API/Term 21 (9_O2T General Purpose Registers 1)/Subterm 25 (9_O2T General Purpose Registers 1)/Outputs/O2T Reg 1[13]
//     PlcTask Outputs/Robot_UR3.UR_inputs/Ints/INT2[2] <-> API/Term 21 (9_O2T General Purpose Registers 1)/Subterm 25 (9_O2T General Purpose Registers 1)/Outputs/O2T Reg 1[14]
//     PlcTask Outputs/Robot_UR3.UR_inputs/Ints/INT2[3] <-> API/Term 21 (9_O2T General Purpose Registers 1)/Subterm 25 (9_O2T General Purpose Registers 1)/Outputs/O2T Reg 1[15]
//     PlcTask Outputs/Robot_UR3.UR_inputs/Ints/INT3[0] <-> API/Term 21 (9_O2T General Purpose Registers 1)/Subterm 25 (9_O2T General Purpose Registers 1)/Outputs/O2T Reg 1[16]
//     PlcTask Outputs/Robot_UR3.UR_inputs/Ints/INT3[1] <-> API/Term 21 (9_O2T General Purpose Registers 1)/Subterm 25 (9_O2T General Purpose Registers 1)/Outputs/O2T Reg 1[17]
//     PlcTask Outputs/Robot_UR3.UR_inputs/Ints/INT3[2] <-> API/Term 21 (9_O2T General Purpose Registers 1)/Subterm 25 (9_O2T General Purpose Registers 1)/Outputs/O2T Reg 1[18]
//     PlcTask Outputs/Robot_UR3.UR_inputs/Ints/INT3[3] <-> API/Term 21 (9_O2T General Purpose Registers 1)/Subterm 25 (9_O2T General Purpose Registers 1)/Outputs/O2T Reg 1[19]
//     PlcTask Outputs/Robot_UR3.UR_inputs/Ints/INT4[0] <-> API/Term 21 (9_O2T General Purpose Registers 1)/Subterm 25 (9_O2T General Purpose Registers 1)/Outputs/O2T Reg 1[20]
//     PlcTask Outputs/Robot_UR3.UR_inputs/Ints/INT4[1] <-> API/Term 21 (9_O2T General Purpose Registers 1)/Subterm 25 (9_O2T General Purpose Registers 1)/Outputs/O2T Reg 1[21]
//     PlcTask Outputs/Robot_UR3.UR_inputs/Ints/INT4[2] <-> API/Term 21 (9_O2T General Purpose Registers 1)/Subterm 25 (9_O2T General Purpose Registers 1)/Outputs/O2T Reg 1[22]
//     PlcTask Outputs/Robot_UR3.UR_inputs/Ints/INT4[3] <-> API/Term 21 (9_O2T General Purpose Registers 1)/Subterm 25 (9_O2T General Purpose Registers 1)/Outputs/O2T Reg 1[23]
//     PlcTask Outputs/Robot_UR3.UR_inputs/Ints/INT5[0] <-> API/Term 21 (9_O2T General Purpose Registers 1)/Subterm 25 (9_O2T General Purpose Registers 1)/Outputs/O2T Reg 1[24]
//     PlcTask Outputs/Robot_UR3.UR_inputs/Ints/INT5[1] <-> API/Term 21 (9_O2T General Purpose Registers 1)/Subterm 25 (9_O2T General Purpose Registers 1)/Outputs/O2T Reg 1[25]
//     PlcTask Outputs/Robot_UR3.UR_inputs/Ints/INT5[2] <-> API/Term 21 (9_O2T General Purpose Registers 1)/Subterm 25 (9_O2T General Purpose Registers 1)/Outputs/O2T Reg 1[26]
//     PlcTask Outputs/Robot_UR3.UR_inputs/Ints/INT5[3] <-> API/Term 21 (9_O2T General Purpose Registers 1)/Subterm 25 (9_O2T General Purpose Registers 1)/Outputs/O2T Reg 1[27]
//     PlcTask Outputs/Robot_UR3.UR_inputs/Ints/INT6[0] <-> API/Term 21 (9_O2T General Purpose Registers 1)/Subterm 25 (9_O2T General Purpose Registers 1)/Outputs/O2T Reg 1[28]
//     PlcTask Outputs/Robot_UR3.UR_inputs/Ints/INT6[1] <-> API/Term 21 (9_O2T General Purpose Registers 1)/Subterm 25 (9_O2T General Purpose Registers 1)/Outputs/O2T Reg 1[29]
//     PlcTask Outputs/Robot_UR3.UR_inputs/Ints/INT6[2] <-> API/Term 21 (9_O2T General Purpose Registers 1)/Subterm 25 (9_O2T General Purpose Registers 1)/Outputs/O2T Reg 1[30]
//     PlcTask Outputs/Robot_UR3.UR_inputs/Ints/INT6[3] <-> API/Term 21 (9_O2T General Purpose Registers 1)/Subterm 25 (9_O2T General Purpose Registers 1)/Outputs/O2T Reg 1[31]
//     PlcTask Outputs/Robot_UR3.UR_inputs/Ints/INT7[0] <-> API/Term 21 (9_O2T General Purpose Registers 1)/Subterm 25 (9_O2T General Purpose Registers 1)/Outputs/O2T Reg 1[32]
//     PlcTask Outputs/Robot_UR3.UR_inputs/Ints/INT7[1] <-> API/Term 21 (9_O2T General Purpose Registers 1)/Subterm 25 (9_O2T General Purpose Registers 1)/Outputs/O2T Reg 1[33]
//     PlcTask Outputs/Robot_UR3.UR_inputs/Ints/INT7[2] <-> API/Term 21 (9_O2T General Purpose Registers 1)/Subterm 25 (9_O2T General Purpose Registers 1)/Outputs/O2T Reg 1[34]
//     PlcTask Outputs/Robot_UR3.UR_inputs/Ints/INT7[3] <-> API/Term 21 (9_O2T General Purpose Registers 1)/Subterm 25 (9_O2T General Purpose Registers 1)/Outputs/O2T Reg 1[35]
//     PlcTask Outputs/Robot_UR3.UR_inputs/Ints/INT8[0] <-> API/Term 21 (9_O2T General Purpose Registers 1)/Subterm 25 (9_O2T General Purpose Registers 1)/Outputs/O2T Reg 1[36]
//     PlcTask Outputs/Robot_UR3.UR_inputs/Ints/INT8[1] <-> API/Term 21 (9_O2T General Purpose Registers 1)/Subterm 25 (9_O2T General Purpose Registers 1)/Outputs/O2T Reg 1[37]
//     PlcTask Outputs/Robot_UR3.UR_inputs/Ints/INT8[2] <-> API/Term 21 (9_O2T General Purpose Registers 1)/Subterm 25 (9_O2T General Purpose Registers 1)/Outputs/O2T Reg 1[38]
//     PlcTask Outputs/Robot_UR3.UR_inputs/Ints/INT8[3] <-> API/Term 21 (9_O2T General Purpose Registers 1)/Subterm 25 (9_O2T General Purpose Registers 1)/Outputs/O2T Reg 1[39]
//     PlcTask Outputs/Robot_UR3.UR_inputs/Ints/INT9[0] <-> API/Term 21 (9_O2T General Purpose Registers 1)/Subterm 25 (9_O2T General Purpose Registers 1)/Outputs/O2T Reg 1[40]
//     PlcTask Outputs/Robot_UR3.UR_inputs/Ints/INT9[1] <-> API/Term 21 (9_O2T General Purpose Registers 1)/Subterm 25 (9_O2T General Purpose Registers 1)/Outputs/O2T Reg 1[41]
//     PlcTask Outputs/Robot_UR3.UR_inputs/Ints/INT9[2] <-> API/Term 21 (9_O2T General Purpose Registers 1)/Subterm 25 (9_O2T General Purpose Registers 1)/Outputs/O2T Reg 1[42]
//     PlcTask Outputs/Robot_UR3.UR_inputs/Ints/INT9[3] <-> API/Term 21 (9_O2T General Purpose Registers 1)/Subterm 25 (9_O2T General Purpose Registers 1)/Outputs/O2T Reg 1[43]
//   p1/p1 Instance <-> Device 4 (EL6631)/uriodev1ur5
//     PlcTask Inputs/Robot_UR5.UR_TCP/FLOAT0[0] <-> API/Term 6 (4_T2O TCP)/Subterm 10 (4_T2O TCP)/Inputs/T2O TCP[0]
//     PlcTask Inputs/Robot_UR5.UR_TCP/FLOAT0[1] <-> API/Term 6 (4_T2O TCP)/Subterm 10 (4_T2O TCP)/Inputs/T2O TCP[1]
//     PlcTask Inputs/Robot_UR5.UR_TCP/FLOAT0[2] <-> API/Term 6 (4_T2O TCP)/Subterm 10 (4_T2O TCP)/Inputs/T2O TCP[2]
//     PlcTask Inputs/Robot_UR5.UR_TCP/FLOAT0[3] <-> API/Term 6 (4_T2O TCP)/Subterm 10 (4_T2O TCP)/Inputs/T2O TCP[3]
//     PlcTask Inputs/Robot_UR5.UR_TCP/FLOAT10[0] <-> API/Term 6 (4_T2O TCP)/Subterm 10 (4_T2O TCP)/Inputs/T2O TCP[40]
//     PlcTask Inputs/Robot_UR5.UR_TCP/FLOAT10[1] <-> API/Term 6 (4_T2O TCP)/Subterm 10 (4_T2O TCP)/Inputs/T2O TCP[41]
//     PlcTask Inputs/Robot_UR5.UR_TCP/FLOAT10[2] <-> API/Term 6 (4_T2O TCP)/Subterm 10 (4_T2O TCP)/Inputs/T2O TCP[42]
//     PlcTask Inputs/Robot_UR5.UR_TCP/FLOAT10[3] <-> API/Term 6 (4_T2O TCP)/Subterm 10 (4_T2O TCP)/Inputs/T2O TCP[43]
//     PlcTask Inputs/Robot_UR5.UR_TCP/FLOAT11[0] <-> API/Term 6 (4_T2O TCP)/Subterm 10 (4_T2O TCP)/Inputs/T2O TCP[44]
//     PlcTask Inputs/Robot_UR5.UR_TCP/FLOAT11[1] <-> API/Term 6 (4_T2O TCP)/Subterm 10 (4_T2O TCP)/Inputs/T2O TCP[45]
//     PlcTask Inputs/Robot_UR5.UR_TCP/FLOAT11[2] <-> API/Term 6 (4_T2O TCP)/Subterm 10 (4_T2O TCP)/Inputs/T2O TCP[46]
//     PlcTask Inputs/Robot_UR5.UR_TCP/FLOAT11[3] <-> API/Term 6 (4_T2O TCP)/Subterm 10 (4_T2O TCP)/Inputs/T2O TCP[47]
//     PlcTask Inputs/Robot_UR5.UR_TCP/FLOAT12[0] <-> API/Term 6 (4_T2O TCP)/Subterm 10 (4_T2O TCP)/Inputs/T2O TCP[48]
//     PlcTask Inputs/Robot_UR5.UR_TCP/FLOAT12[1] <-> API/Term 6 (4_T2O TCP)/Subterm 10 (4_T2O TCP)/Inputs/T2O TCP[49]
//     PlcTask Inputs/Robot_UR5.UR_TCP/FLOAT12[2] <-> API/Term 6 (4_T2O TCP)/Subterm 10 (4_T2O TCP)/Inputs/T2O TCP[50]
//     PlcTask Inputs/Robot_UR5.UR_TCP/FLOAT12[3] <-> API/Term 6 (4_T2O TCP)/Subterm 10 (4_T2O TCP)/Inputs/T2O TCP[51]
//     PlcTask Inputs/Robot_UR5.UR_TCP/FLOAT13[0] <-> API/Term 6 (4_T2O TCP)/Subterm 10 (4_T2O TCP)/Inputs/T2O TCP[52]
//     PlcTask Inputs/Robot_UR5.UR_TCP/FLOAT13[1] <-> API/Term 6 (4_T2O TCP)/Subterm 10 (4_T2O TCP)/Inputs/T2O TCP[53]
//     PlcTask Inputs/Robot_UR5.UR_TCP/FLOAT13[2] <-> API/Term 6 (4_T2O TCP)/Subterm 10 (4_T2O TCP)/Inputs/T2O TCP[54]
//     PlcTask Inputs/Robot_UR5.UR_TCP/FLOAT13[3] <-> API/Term 6 (4_T2O TCP)/Subterm 10 (4_T2O TCP)/Inputs/T2O TCP[55]
//     PlcTask Inputs/Robot_UR5.UR_TCP/FLOAT14[0] <-> API/Term 6 (4_T2O TCP)/Subterm 10 (4_T2O TCP)/Inputs/T2O TCP[56]
//     PlcTask Inputs/Robot_UR5.UR_TCP/FLOAT14[1] <-> API/Term 6 (4_T2O TCP)/Subterm 10 (4_T2O TCP)/Inputs/T2O TCP[57]
//     PlcTask Inputs/Robot_UR5.UR_TCP/FLOAT14[2] <-> API/Term 6 (4_T2O TCP)/Subterm 10 (4_T2O TCP)/Inputs/T2O TCP[58]
//     PlcTask Inputs/Robot_UR5.UR_TCP/FLOAT14[3] <-> API/Term 6 (4_T2O TCP)/Subterm 10 (4_T2O TCP)/Inputs/T2O TCP[59]
//     PlcTask Inputs/Robot_UR5.UR_TCP/FLOAT15[0] <-> API/Term 6 (4_T2O TCP)/Subterm 10 (4_T2O TCP)/Inputs/T2O TCP[60]
//     PlcTask Inputs/Robot_UR5.UR_TCP/FLOAT15[1] <-> API/Term 6 (4_T2O TCP)/Subterm 10 (4_T2O TCP)/Inputs/T2O TCP[61]
//     PlcTask Inputs/Robot_UR5.UR_TCP/FLOAT15[2] <-> API/Term 6 (4_T2O TCP)/Subterm 10 (4_T2O TCP)/Inputs/T2O TCP[62]
//     PlcTask Inputs/Robot_UR5.UR_TCP/FLOAT15[3] <-> API/Term 6 (4_T2O TCP)/Subterm 10 (4_T2O TCP)/Inputs/T2O TCP[63]
//     PlcTask Inputs/Robot_UR5.UR_TCP/FLOAT16[0] <-> API/Term 6 (4_T2O TCP)/Subterm 10 (4_T2O TCP)/Inputs/T2O TCP[64]
//     PlcTask Inputs/Robot_UR5.UR_TCP/FLOAT16[1] <-> API/Term 6 (4_T2O TCP)/Subterm 10 (4_T2O TCP)/Inputs/T2O TCP[65]
//     PlcTask Inputs/Robot_UR5.UR_TCP/FLOAT16[2] <-> API/Term 6 (4_T2O TCP)/Subterm 10 (4_T2O TCP)/Inputs/T2O TCP[66]
//     PlcTask Inputs/Robot_UR5.UR_TCP/FLOAT16[3] <-> API/Term 6 (4_T2O TCP)/Subterm 10 (4_T2O TCP)/Inputs/T2O TCP[67]
//     PlcTask Inputs/Robot_UR5.UR_TCP/FLOAT17[0] <-> API/Term 6 (4_T2O TCP)/Subterm 10 (4_T2O TCP)/Inputs/T2O TCP[68]
//     PlcTask Inputs/Robot_UR5.UR_TCP/FLOAT17[1] <-> API/Term 6 (4_T2O TCP)/Subterm 10 (4_T2O TCP)/Inputs/T2O TCP[69]
//     PlcTask Inputs/Robot_UR5.UR_TCP/FLOAT17[2] <-> API/Term 6 (4_T2O TCP)/Subterm 10 (4_T2O TCP)/Inputs/T2O TCP[70]
//     PlcTask Inputs/Robot_UR5.UR_TCP/FLOAT17[3] <-> API/Term 6 (4_T2O TCP)/Subterm 10 (4_T2O TCP)/Inputs/T2O TCP[71]
//     PlcTask Inputs/Robot_UR5.UR_TCP/FLOAT18[0] <-> API/Term 6 (4_T2O TCP)/Subterm 10 (4_T2O TCP)/Inputs/T2O TCP[68]
//     PlcTask Inputs/Robot_UR5.UR_TCP/FLOAT18[1] <-> API/Term 6 (4_T2O TCP)/Subterm 10 (4_T2O TCP)/Inputs/T2O TCP[72]
//     PlcTask Inputs/Robot_UR5.UR_TCP/FLOAT18[2] <-> API/Term 6 (4_T2O TCP)/Subterm 10 (4_T2O TCP)/Inputs/T2O TCP[73]
//     PlcTask Inputs/Robot_UR5.UR_TCP/FLOAT18[3] <-> API/Term 6 (4_T2O TCP)/Subterm 10 (4_T2O TCP)/Inputs/T2O TCP[74]
//     PlcTask Inputs/Robot_UR5.UR_TCP/FLOAT1[0] <-> API/Term 6 (4_T2O TCP)/Subterm 10 (4_T2O TCP)/Inputs/T2O TCP[4]
//     PlcTask Inputs/Robot_UR5.UR_TCP/FLOAT1[1] <-> API/Term 6 (4_T2O TCP)/Subterm 10 (4_T2O TCP)/Inputs/T2O TCP[5]
//     PlcTask Inputs/Robot_UR5.UR_TCP/FLOAT1[2] <-> API/Term 6 (4_T2O TCP)/Subterm 10 (4_T2O TCP)/Inputs/T2O TCP[6]
//     PlcTask Inputs/Robot_UR5.UR_TCP/FLOAT1[3] <-> API/Term 6 (4_T2O TCP)/Subterm 10 (4_T2O TCP)/Inputs/T2O TCP[7]
//     PlcTask Inputs/Robot_UR5.UR_TCP/FLOAT2[0] <-> API/Term 6 (4_T2O TCP)/Subterm 10 (4_T2O TCP)/Inputs/T2O TCP[8]
//     PlcTask Inputs/Robot_UR5.UR_TCP/FLOAT2[1] <-> API/Term 6 (4_T2O TCP)/Subterm 10 (4_T2O TCP)/Inputs/T2O TCP[9]
//     PlcTask Inputs/Robot_UR5.UR_TCP/FLOAT2[2] <-> API/Term 6 (4_T2O TCP)/Subterm 10 (4_T2O TCP)/Inputs/T2O TCP[10]
//     PlcTask Inputs/Robot_UR5.UR_TCP/FLOAT2[3] <-> API/Term 6 (4_T2O TCP)/Subterm 10 (4_T2O TCP)/Inputs/T2O TCP[11]
//     PlcTask Inputs/Robot_UR5.UR_TCP/FLOAT3[0] <-> API/Term 6 (4_T2O TCP)/Subterm 10 (4_T2O TCP)/Inputs/T2O TCP[12]
//     PlcTask Inputs/Robot_UR5.UR_TCP/FLOAT3[1] <-> API/Term 6 (4_T2O TCP)/Subterm 10 (4_T2O TCP)/Inputs/T2O TCP[13]
//     PlcTask Inputs/Robot_UR5.UR_TCP/FLOAT3[2] <-> API/Term 6 (4_T2O TCP)/Subterm 10 (4_T2O TCP)/Inputs/T2O TCP[14]
//     PlcTask Inputs/Robot_UR5.UR_TCP/FLOAT3[3] <-> API/Term 6 (4_T2O TCP)/Subterm 10 (4_T2O TCP)/Inputs/T2O TCP[15]
//     PlcTask Inputs/Robot_UR5.UR_TCP/FLOAT4[0] <-> API/Term 6 (4_T2O TCP)/Subterm 10 (4_T2O TCP)/Inputs/T2O TCP[16]
//     PlcTask Inputs/Robot_UR5.UR_TCP/FLOAT4[1] <-> API/Term 6 (4_T2O TCP)/Subterm 10 (4_T2O TCP)/Inputs/T2O TCP[17]
//     PlcTask Inputs/Robot_UR5.UR_TCP/FLOAT4[2] <-> API/Term 6 (4_T2O TCP)/Subterm 10 (4_T2O TCP)/Inputs/T2O TCP[18]
//     PlcTask Inputs/Robot_UR5.UR_TCP/FLOAT4[3] <-> API/Term 6 (4_T2O TCP)/Subterm 10 (4_T2O TCP)/Inputs/T2O TCP[19]
//     PlcTask Inputs/Robot_UR5.UR_TCP/FLOAT5[0] <-> API/Term 6 (4_T2O TCP)/Subterm 10 (4_T2O TCP)/Inputs/T2O TCP[20]
//     PlcTask Inputs/Robot_UR5.UR_TCP/FLOAT5[1] <-> API/Term 6 (4_T2O TCP)/Subterm 10 (4_T2O TCP)/Inputs/T2O TCP[21]
//     PlcTask Inputs/Robot_UR5.UR_TCP/FLOAT5[2] <-> API/Term 6 (4_T2O TCP)/Subterm 10 (4_T2O TCP)/Inputs/T2O TCP[22]
//     PlcTask Inputs/Robot_UR5.UR_TCP/FLOAT5[3] <-> API/Term 6 (4_T2O TCP)/Subterm 10 (4_T2O TCP)/Inputs/T2O TCP[23]
//     PlcTask Inputs/Robot_UR5.UR_TCP/FLOAT6[0] <-> API/Term 6 (4_T2O TCP)/Subterm 10 (4_T2O TCP)/Inputs/T2O TCP[24]
//     PlcTask Inputs/Robot_UR5.UR_TCP/FLOAT6[1] <-> API/Term 6 (4_T2O TCP)/Subterm 10 (4_T2O TCP)/Inputs/T2O TCP[25]
//     PlcTask Inputs/Robot_UR5.UR_TCP/FLOAT6[2] <-> API/Term 6 (4_T2O TCP)/Subterm 10 (4_T2O TCP)/Inputs/T2O TCP[26]
//     PlcTask Inputs/Robot_UR5.UR_TCP/FLOAT6[3] <-> API/Term 6 (4_T2O TCP)/Subterm 10 (4_T2O TCP)/Inputs/T2O TCP[27]
//     PlcTask Inputs/Robot_UR5.UR_TCP/FLOAT7[0] <-> API/Term 6 (4_T2O TCP)/Subterm 10 (4_T2O TCP)/Inputs/T2O TCP[28]
//     PlcTask Inputs/Robot_UR5.UR_TCP/FLOAT7[1] <-> API/Term 6 (4_T2O TCP)/Subterm 10 (4_T2O TCP)/Inputs/T2O TCP[29]
//     PlcTask Inputs/Robot_UR5.UR_TCP/FLOAT7[2] <-> API/Term 6 (4_T2O TCP)/Subterm 10 (4_T2O TCP)/Inputs/T2O TCP[30]
//     PlcTask Inputs/Robot_UR5.UR_TCP/FLOAT7[3] <-> API/Term 6 (4_T2O TCP)/Subterm 10 (4_T2O TCP)/Inputs/T2O TCP[31]
//     PlcTask Inputs/Robot_UR5.UR_TCP/FLOAT8[0] <-> API/Term 6 (4_T2O TCP)/Subterm 10 (4_T2O TCP)/Inputs/T2O TCP[32]
//     PlcTask Inputs/Robot_UR5.UR_TCP/FLOAT8[1] <-> API/Term 6 (4_T2O TCP)/Subterm 10 (4_T2O TCP)/Inputs/T2O TCP[33]
//     PlcTask Inputs/Robot_UR5.UR_TCP/FLOAT8[2] <-> API/Term 6 (4_T2O TCP)/Subterm 10 (4_T2O TCP)/Inputs/T2O TCP[34]
//     PlcTask Inputs/Robot_UR5.UR_TCP/FLOAT8[3] <-> API/Term 6 (4_T2O TCP)/Subterm 10 (4_T2O TCP)/Inputs/T2O TCP[35]
//     PlcTask Inputs/Robot_UR5.UR_TCP/FLOAT9[0] <-> API/Term 6 (4_T2O TCP)/Subterm 10 (4_T2O TCP)/Inputs/T2O TCP[36]
//     PlcTask Inputs/Robot_UR5.UR_TCP/FLOAT9[1] <-> API/Term 6 (4_T2O TCP)/Subterm 10 (4_T2O TCP)/Inputs/T2O TCP[37]
//     PlcTask Inputs/Robot_UR5.UR_TCP/FLOAT9[2] <-> API/Term 6 (4_T2O TCP)/Subterm 10 (4_T2O TCP)/Inputs/T2O TCP[38]
//     PlcTask Inputs/Robot_UR5.UR_TCP/FLOAT9[3] <-> API/Term 6 (4_T2O TCP)/Subterm 10 (4_T2O TCP)/Inputs/T2O TCP[39]
//     PlcTask Inputs/Robot_UR5.UR_outputs/B{0..56 step 8} <-> API/Term 7 (5_T2O General Purpose Bit Registers)/Subterm 11 (5_T2O General Purpose Bit Registers)/Inputs/T2O Bit Registers[{0..7}]  (8 links)
//     PlcTask Inputs/Robot_UR5.UR_outputs/B1 <-> API/Term 7 (5_T2O General Purpose Bit Registers)/Subterm 11 (5_T2O General Purpose Bit Registers)/Inputs/T2O Bit Registers[0] @bit 1
//     PlcTask Inputs/Robot_UR5.UR_outputs/B10 <-> API/Term 7 (5_T2O General Purpose Bit Registers)/Subterm 11 (5_T2O General Purpose Bit Registers)/Inputs/T2O Bit Registers[1] @bit 2
//     PlcTask Inputs/Robot_UR5.UR_outputs/B11 <-> API/Term 7 (5_T2O General Purpose Bit Registers)/Subterm 11 (5_T2O General Purpose Bit Registers)/Inputs/T2O Bit Registers[1] @bit 3
//     PlcTask Inputs/Robot_UR5.UR_outputs/B12 <-> API/Term 7 (5_T2O General Purpose Bit Registers)/Subterm 11 (5_T2O General Purpose Bit Registers)/Inputs/T2O Bit Registers[1] @bit 4
//     PlcTask Inputs/Robot_UR5.UR_outputs/B13 <-> API/Term 7 (5_T2O General Purpose Bit Registers)/Subterm 11 (5_T2O General Purpose Bit Registers)/Inputs/T2O Bit Registers[1] @bit 5
//     PlcTask Inputs/Robot_UR5.UR_outputs/B14 <-> API/Term 7 (5_T2O General Purpose Bit Registers)/Subterm 11 (5_T2O General Purpose Bit Registers)/Inputs/T2O Bit Registers[1] @bit 6
//     PlcTask Inputs/Robot_UR5.UR_outputs/B15 <-> API/Term 7 (5_T2O General Purpose Bit Registers)/Subterm 11 (5_T2O General Purpose Bit Registers)/Inputs/T2O Bit Registers[1] @bit 7
//     PlcTask Inputs/Robot_UR5.UR_outputs/B17 <-> API/Term 7 (5_T2O General Purpose Bit Registers)/Subterm 11 (5_T2O General Purpose Bit Registers)/Inputs/T2O Bit Registers[2] @bit 1
//     PlcTask Inputs/Robot_UR5.UR_outputs/B18 <-> API/Term 7 (5_T2O General Purpose Bit Registers)/Subterm 11 (5_T2O General Purpose Bit Registers)/Inputs/T2O Bit Registers[2] @bit 2
//     PlcTask Inputs/Robot_UR5.UR_outputs/B19 <-> API/Term 7 (5_T2O General Purpose Bit Registers)/Subterm 11 (5_T2O General Purpose Bit Registers)/Inputs/T2O Bit Registers[2] @bit 3
//     PlcTask Inputs/Robot_UR5.UR_outputs/B2 <-> API/Term 7 (5_T2O General Purpose Bit Registers)/Subterm 11 (5_T2O General Purpose Bit Registers)/Inputs/T2O Bit Registers[0] @bit 2
//     PlcTask Inputs/Robot_UR5.UR_outputs/B20 <-> API/Term 7 (5_T2O General Purpose Bit Registers)/Subterm 11 (5_T2O General Purpose Bit Registers)/Inputs/T2O Bit Registers[2] @bit 4
//     PlcTask Inputs/Robot_UR5.UR_outputs/B21 <-> API/Term 7 (5_T2O General Purpose Bit Registers)/Subterm 11 (5_T2O General Purpose Bit Registers)/Inputs/T2O Bit Registers[2] @bit 5
//     PlcTask Inputs/Robot_UR5.UR_outputs/B22 <-> API/Term 7 (5_T2O General Purpose Bit Registers)/Subterm 11 (5_T2O General Purpose Bit Registers)/Inputs/T2O Bit Registers[2] @bit 6
//     PlcTask Inputs/Robot_UR5.UR_outputs/B23 <-> API/Term 7 (5_T2O General Purpose Bit Registers)/Subterm 11 (5_T2O General Purpose Bit Registers)/Inputs/T2O Bit Registers[2] @bit 7
//     PlcTask Inputs/Robot_UR5.UR_outputs/B25 <-> API/Term 7 (5_T2O General Purpose Bit Registers)/Subterm 11 (5_T2O General Purpose Bit Registers)/Inputs/T2O Bit Registers[3] @bit 1
//     PlcTask Inputs/Robot_UR5.UR_outputs/B26 <-> API/Term 7 (5_T2O General Purpose Bit Registers)/Subterm 11 (5_T2O General Purpose Bit Registers)/Inputs/T2O Bit Registers[3] @bit 2
//     PlcTask Inputs/Robot_UR5.UR_outputs/B27 <-> API/Term 7 (5_T2O General Purpose Bit Registers)/Subterm 11 (5_T2O General Purpose Bit Registers)/Inputs/T2O Bit Registers[3] @bit 3
//     PlcTask Inputs/Robot_UR5.UR_outputs/B28 <-> API/Term 7 (5_T2O General Purpose Bit Registers)/Subterm 11 (5_T2O General Purpose Bit Registers)/Inputs/T2O Bit Registers[3] @bit 4
//     PlcTask Inputs/Robot_UR5.UR_outputs/B29 <-> API/Term 7 (5_T2O General Purpose Bit Registers)/Subterm 11 (5_T2O General Purpose Bit Registers)/Inputs/T2O Bit Registers[3] @bit 5
//     PlcTask Inputs/Robot_UR5.UR_outputs/B3 <-> API/Term 7 (5_T2O General Purpose Bit Registers)/Subterm 11 (5_T2O General Purpose Bit Registers)/Inputs/T2O Bit Registers[0] @bit 3
//     PlcTask Inputs/Robot_UR5.UR_outputs/B30 <-> API/Term 7 (5_T2O General Purpose Bit Registers)/Subterm 11 (5_T2O General Purpose Bit Registers)/Inputs/T2O Bit Registers[3] @bit 6
//     PlcTask Inputs/Robot_UR5.UR_outputs/B31 <-> API/Term 7 (5_T2O General Purpose Bit Registers)/Subterm 11 (5_T2O General Purpose Bit Registers)/Inputs/T2O Bit Registers[3] @bit 7
//     PlcTask Inputs/Robot_UR5.UR_outputs/B33 <-> API/Term 7 (5_T2O General Purpose Bit Registers)/Subterm 11 (5_T2O General Purpose Bit Registers)/Inputs/T2O Bit Registers[4] @bit 1
//     PlcTask Inputs/Robot_UR5.UR_outputs/B34 <-> API/Term 7 (5_T2O General Purpose Bit Registers)/Subterm 11 (5_T2O General Purpose Bit Registers)/Inputs/T2O Bit Registers[4] @bit 2
//     PlcTask Inputs/Robot_UR5.UR_outputs/B35 <-> API/Term 7 (5_T2O General Purpose Bit Registers)/Subterm 11 (5_T2O General Purpose Bit Registers)/Inputs/T2O Bit Registers[4] @bit 3
//     PlcTask Inputs/Robot_UR5.UR_outputs/B36 <-> API/Term 7 (5_T2O General Purpose Bit Registers)/Subterm 11 (5_T2O General Purpose Bit Registers)/Inputs/T2O Bit Registers[4] @bit 4
//     PlcTask Inputs/Robot_UR5.UR_outputs/B37 <-> API/Term 7 (5_T2O General Purpose Bit Registers)/Subterm 11 (5_T2O General Purpose Bit Registers)/Inputs/T2O Bit Registers[4] @bit 5
//     PlcTask Inputs/Robot_UR5.UR_outputs/B38 <-> API/Term 7 (5_T2O General Purpose Bit Registers)/Subterm 11 (5_T2O General Purpose Bit Registers)/Inputs/T2O Bit Registers[4] @bit 6
//     PlcTask Inputs/Robot_UR5.UR_outputs/B39 <-> API/Term 7 (5_T2O General Purpose Bit Registers)/Subterm 11 (5_T2O General Purpose Bit Registers)/Inputs/T2O Bit Registers[4] @bit 7
//     PlcTask Inputs/Robot_UR5.UR_outputs/B4 <-> API/Term 7 (5_T2O General Purpose Bit Registers)/Subterm 11 (5_T2O General Purpose Bit Registers)/Inputs/T2O Bit Registers[0] @bit 4
//     PlcTask Inputs/Robot_UR5.UR_outputs/B41 <-> API/Term 7 (5_T2O General Purpose Bit Registers)/Subterm 11 (5_T2O General Purpose Bit Registers)/Inputs/T2O Bit Registers[5] @bit 1
//     PlcTask Inputs/Robot_UR5.UR_outputs/B42 <-> API/Term 7 (5_T2O General Purpose Bit Registers)/Subterm 11 (5_T2O General Purpose Bit Registers)/Inputs/T2O Bit Registers[5] @bit 2
//     PlcTask Inputs/Robot_UR5.UR_outputs/B43 <-> API/Term 7 (5_T2O General Purpose Bit Registers)/Subterm 11 (5_T2O General Purpose Bit Registers)/Inputs/T2O Bit Registers[5] @bit 3
//     PlcTask Inputs/Robot_UR5.UR_outputs/B44 <-> API/Term 7 (5_T2O General Purpose Bit Registers)/Subterm 11 (5_T2O General Purpose Bit Registers)/Inputs/T2O Bit Registers[5] @bit 4
//     PlcTask Inputs/Robot_UR5.UR_outputs/B45 <-> API/Term 7 (5_T2O General Purpose Bit Registers)/Subterm 11 (5_T2O General Purpose Bit Registers)/Inputs/T2O Bit Registers[5] @bit 5
//     PlcTask Inputs/Robot_UR5.UR_outputs/B46 <-> API/Term 7 (5_T2O General Purpose Bit Registers)/Subterm 11 (5_T2O General Purpose Bit Registers)/Inputs/T2O Bit Registers[5] @bit 6
//     PlcTask Inputs/Robot_UR5.UR_outputs/B47 <-> API/Term 7 (5_T2O General Purpose Bit Registers)/Subterm 11 (5_T2O General Purpose Bit Registers)/Inputs/T2O Bit Registers[5] @bit 7
//     PlcTask Inputs/Robot_UR5.UR_outputs/B49 <-> API/Term 7 (5_T2O General Purpose Bit Registers)/Subterm 11 (5_T2O General Purpose Bit Registers)/Inputs/T2O Bit Registers[6] @bit 1
//     PlcTask Inputs/Robot_UR5.UR_outputs/B5 <-> API/Term 7 (5_T2O General Purpose Bit Registers)/Subterm 11 (5_T2O General Purpose Bit Registers)/Inputs/T2O Bit Registers[0] @bit 5
//     PlcTask Inputs/Robot_UR5.UR_outputs/B50 <-> API/Term 7 (5_T2O General Purpose Bit Registers)/Subterm 11 (5_T2O General Purpose Bit Registers)/Inputs/T2O Bit Registers[6] @bit 2
//     PlcTask Inputs/Robot_UR5.UR_outputs/B51 <-> API/Term 7 (5_T2O General Purpose Bit Registers)/Subterm 11 (5_T2O General Purpose Bit Registers)/Inputs/T2O Bit Registers[6] @bit 3
//     PlcTask Inputs/Robot_UR5.UR_outputs/B52 <-> API/Term 7 (5_T2O General Purpose Bit Registers)/Subterm 11 (5_T2O General Purpose Bit Registers)/Inputs/T2O Bit Registers[6] @bit 4
//     PlcTask Inputs/Robot_UR5.UR_outputs/B53 <-> API/Term 7 (5_T2O General Purpose Bit Registers)/Subterm 11 (5_T2O General Purpose Bit Registers)/Inputs/T2O Bit Registers[6] @bit 5
//     PlcTask Inputs/Robot_UR5.UR_outputs/B54 <-> API/Term 7 (5_T2O General Purpose Bit Registers)/Subterm 11 (5_T2O General Purpose Bit Registers)/Inputs/T2O Bit Registers[6] @bit 6
//     PlcTask Inputs/Robot_UR5.UR_outputs/B55 <-> API/Term 7 (5_T2O General Purpose Bit Registers)/Subterm 11 (5_T2O General Purpose Bit Registers)/Inputs/T2O Bit Registers[6] @bit 7
//     PlcTask Inputs/Robot_UR5.UR_outputs/B57 <-> API/Term 7 (5_T2O General Purpose Bit Registers)/Subterm 11 (5_T2O General Purpose Bit Registers)/Inputs/T2O Bit Registers[7] @bit 1
//     PlcTask Inputs/Robot_UR5.UR_outputs/B58 <-> API/Term 7 (5_T2O General Purpose Bit Registers)/Subterm 11 (5_T2O General Purpose Bit Registers)/Inputs/T2O Bit Registers[7] @bit 2
//     PlcTask Inputs/Robot_UR5.UR_outputs/B59 <-> API/Term 7 (5_T2O General Purpose Bit Registers)/Subterm 11 (5_T2O General Purpose Bit Registers)/Inputs/T2O Bit Registers[7] @bit 3
//     PlcTask Inputs/Robot_UR5.UR_outputs/B6 <-> API/Term 7 (5_T2O General Purpose Bit Registers)/Subterm 11 (5_T2O General Purpose Bit Registers)/Inputs/T2O Bit Registers[0] @bit 6
//     PlcTask Inputs/Robot_UR5.UR_outputs/B60 <-> API/Term 7 (5_T2O General Purpose Bit Registers)/Subterm 11 (5_T2O General Purpose Bit Registers)/Inputs/T2O Bit Registers[7] @bit 4
//     PlcTask Inputs/Robot_UR5.UR_outputs/B61 <-> API/Term 7 (5_T2O General Purpose Bit Registers)/Subterm 11 (5_T2O General Purpose Bit Registers)/Inputs/T2O Bit Registers[7] @bit 5
//     PlcTask Inputs/Robot_UR5.UR_outputs/B62 <-> API/Term 7 (5_T2O General Purpose Bit Registers)/Subterm 11 (5_T2O General Purpose Bit Registers)/Inputs/T2O Bit Registers[7] @bit 6
//     PlcTask Inputs/Robot_UR5.UR_outputs/B63 <-> API/Term 7 (5_T2O General Purpose Bit Registers)/Subterm 11 (5_T2O General Purpose Bit Registers)/Inputs/T2O Bit Registers[7] @bit 7
//     PlcTask Inputs/Robot_UR5.UR_outputs/B7 <-> API/Term 7 (5_T2O General Purpose Bit Registers)/Subterm 11 (5_T2O General Purpose Bit Registers)/Inputs/T2O Bit Registers[0] @bit 7
//     PlcTask Inputs/Robot_UR5.UR_outputs/B9 <-> API/Term 7 (5_T2O General Purpose Bit Registers)/Subterm 11 (5_T2O General Purpose Bit Registers)/Inputs/T2O Bit Registers[1] @bit 1
//     PlcTask Inputs/Robot_UR5.UR_outputs_int/INT0[0] <-> API/Term 8 (6_T2O General Purpose Int Registers)/Subterm 12 (6_T2O General Purpose Int Registers)/Inputs/T2O Int Registers[0]
//     PlcTask Inputs/Robot_UR5.UR_outputs_int/INT0[1] <-> API/Term 8 (6_T2O General Purpose Int Registers)/Subterm 12 (6_T2O General Purpose Int Registers)/Inputs/T2O Int Registers[1]
//     PlcTask Inputs/Robot_UR5.UR_outputs_int/INT0[2] <-> API/Term 8 (6_T2O General Purpose Int Registers)/Subterm 12 (6_T2O General Purpose Int Registers)/Inputs/T2O Int Registers[2]
//     PlcTask Inputs/Robot_UR5.UR_outputs_int/INT0[3] <-> API/Term 8 (6_T2O General Purpose Int Registers)/Subterm 12 (6_T2O General Purpose Int Registers)/Inputs/T2O Int Registers[3]
//     PlcTask Inputs/Robot_UR5.UR_outputs_int/INT1[0] <-> API/Term 8 (6_T2O General Purpose Int Registers)/Subterm 12 (6_T2O General Purpose Int Registers)/Inputs/T2O Int Registers[4]
//     PlcTask Inputs/Robot_UR5.UR_outputs_int/INT1[1] <-> API/Term 8 (6_T2O General Purpose Int Registers)/Subterm 12 (6_T2O General Purpose Int Registers)/Inputs/T2O Int Registers[5]
//     PlcTask Inputs/Robot_UR5.UR_outputs_int/INT1[2] <-> API/Term 8 (6_T2O General Purpose Int Registers)/Subterm 12 (6_T2O General Purpose Int Registers)/Inputs/T2O Int Registers[6]
//     PlcTask Inputs/Robot_UR5.UR_outputs_int/INT1[3] <-> API/Term 8 (6_T2O General Purpose Int Registers)/Subterm 12 (6_T2O General Purpose Int Registers)/Inputs/T2O Int Registers[7]
//     PlcTask Inputs/Robot_UR5.UR_outputs_int/INT2[0] <-> API/Term 8 (6_T2O General Purpose Int Registers)/Subterm 12 (6_T2O General Purpose Int Registers)/Inputs/T2O Int Registers[8]
//     PlcTask Inputs/Robot_UR5.UR_outputs_int/INT2[1] <-> API/Term 8 (6_T2O General Purpose Int Registers)/Subterm 12 (6_T2O General Purpose Int Registers)/Inputs/T2O Int Registers[9]
//     PlcTask Inputs/Robot_UR5.UR_outputs_int/INT2[2] <-> API/Term 8 (6_T2O General Purpose Int Registers)/Subterm 12 (6_T2O General Purpose Int Registers)/Inputs/T2O Int Registers[10]
//     PlcTask Inputs/Robot_UR5.UR_outputs_int/INT2[3] <-> API/Term 8 (6_T2O General Purpose Int Registers)/Subterm 12 (6_T2O General Purpose Int Registers)/Inputs/T2O Int Registers[11]
//     PlcTask Inputs/Robot_UR5.UR_outputs_int/INT3[0] <-> API/Term 8 (6_T2O General Purpose Int Registers)/Subterm 12 (6_T2O General Purpose Int Registers)/Inputs/T2O Int Registers[12]
//     PlcTask Inputs/Robot_UR5.UR_outputs_int/INT3[1] <-> API/Term 8 (6_T2O General Purpose Int Registers)/Subterm 12 (6_T2O General Purpose Int Registers)/Inputs/T2O Int Registers[13]
//     PlcTask Inputs/Robot_UR5.UR_outputs_int/INT3[2] <-> API/Term 8 (6_T2O General Purpose Int Registers)/Subterm 12 (6_T2O General Purpose Int Registers)/Inputs/T2O Int Registers[14]
//     PlcTask Inputs/Robot_UR5.UR_outputs_int/INT3[3] <-> API/Term 8 (6_T2O General Purpose Int Registers)/Subterm 12 (6_T2O General Purpose Int Registers)/Inputs/T2O Int Registers[15]
//     PlcTask Inputs/Robot_UR5.UR_outputs_int/INT4[0] <-> API/Term 8 (6_T2O General Purpose Int Registers)/Subterm 12 (6_T2O General Purpose Int Registers)/Inputs/T2O Int Registers[16]
//     PlcTask Inputs/Robot_UR5.UR_outputs_int/INT4[1] <-> API/Term 8 (6_T2O General Purpose Int Registers)/Subterm 12 (6_T2O General Purpose Int Registers)/Inputs/T2O Int Registers[17]
//     PlcTask Inputs/Robot_UR5.UR_outputs_int/INT4[2] <-> API/Term 8 (6_T2O General Purpose Int Registers)/Subterm 12 (6_T2O General Purpose Int Registers)/Inputs/T2O Int Registers[18]
//     PlcTask Inputs/Robot_UR5.UR_outputs_int/INT4[3] <-> API/Term 8 (6_T2O General Purpose Int Registers)/Subterm 12 (6_T2O General Purpose Int Registers)/Inputs/T2O Int Registers[19]
//     PlcTask Inputs/Robot_UR5.UR_outputs_int/INT5[0] <-> API/Term 8 (6_T2O General Purpose Int Registers)/Subterm 12 (6_T2O General Purpose Int Registers)/Inputs/T2O Int Registers[20]
//     PlcTask Inputs/Robot_UR5.UR_outputs_int/INT5[1] <-> API/Term 8 (6_T2O General Purpose Int Registers)/Subterm 12 (6_T2O General Purpose Int Registers)/Inputs/T2O Int Registers[21]
//     PlcTask Inputs/Robot_UR5.UR_outputs_int/INT5[2] <-> API/Term 8 (6_T2O General Purpose Int Registers)/Subterm 12 (6_T2O General Purpose Int Registers)/Inputs/T2O Int Registers[22]
//     PlcTask Inputs/Robot_UR5.UR_outputs_int/INT5[3] <-> API/Term 8 (6_T2O General Purpose Int Registers)/Subterm 12 (6_T2O General Purpose Int Registers)/Inputs/T2O Int Registers[23]
//     PlcTask Inputs/Robot_UR5.UR_outputs_int/INT6[0] <-> API/Term 8 (6_T2O General Purpose Int Registers)/Subterm 12 (6_T2O General Purpose Int Registers)/Inputs/T2O Int Registers[24]
//     PlcTask Inputs/Robot_UR5.UR_outputs_int/INT6[1] <-> API/Term 8 (6_T2O General Purpose Int Registers)/Subterm 12 (6_T2O General Purpose Int Registers)/Inputs/T2O Int Registers[25]
//     PlcTask Inputs/Robot_UR5.UR_outputs_int/INT6[2] <-> API/Term 8 (6_T2O General Purpose Int Registers)/Subterm 12 (6_T2O General Purpose Int Registers)/Inputs/T2O Int Registers[26]
//     PlcTask Inputs/Robot_UR5.UR_outputs_int/INT6[3] <-> API/Term 8 (6_T2O General Purpose Int Registers)/Subterm 12 (6_T2O General Purpose Int Registers)/Inputs/T2O Int Registers[27]
//     PlcTask Outputs/Robot_UR5.UR_inputs/Bits/B{0..24 step 8} <-> API/Term 11 (9_O2T General Purpose Registers 1)/Subterm 15 (9_O2T General Purpose Registers 1)/Outputs/O2T Reg 1[{0..3}]  (4 links)
//     PlcTask Outputs/Robot_UR5.UR_inputs/Bits/B1 <-> API/Term 11 (9_O2T General Purpose Registers 1)/Subterm 15 (9_O2T General Purpose Registers 1)/Outputs/O2T Reg 1[0] @bit 1
//     PlcTask Outputs/Robot_UR5.UR_inputs/Bits/B10 <-> API/Term 11 (9_O2T General Purpose Registers 1)/Subterm 15 (9_O2T General Purpose Registers 1)/Outputs/O2T Reg 1[1] @bit 2
//     PlcTask Outputs/Robot_UR5.UR_inputs/Bits/B11 <-> API/Term 11 (9_O2T General Purpose Registers 1)/Subterm 15 (9_O2T General Purpose Registers 1)/Outputs/O2T Reg 1[1] @bit 3
//     PlcTask Outputs/Robot_UR5.UR_inputs/Bits/B12 <-> API/Term 11 (9_O2T General Purpose Registers 1)/Subterm 15 (9_O2T General Purpose Registers 1)/Outputs/O2T Reg 1[1] @bit 4
//     PlcTask Outputs/Robot_UR5.UR_inputs/Bits/B13 <-> API/Term 11 (9_O2T General Purpose Registers 1)/Subterm 15 (9_O2T General Purpose Registers 1)/Outputs/O2T Reg 1[1] @bit 5
//     PlcTask Outputs/Robot_UR5.UR_inputs/Bits/B14 <-> API/Term 11 (9_O2T General Purpose Registers 1)/Subterm 15 (9_O2T General Purpose Registers 1)/Outputs/O2T Reg 1[1] @bit 6
//     PlcTask Outputs/Robot_UR5.UR_inputs/Bits/B15 <-> API/Term 11 (9_O2T General Purpose Registers 1)/Subterm 15 (9_O2T General Purpose Registers 1)/Outputs/O2T Reg 1[1] @bit 7
//     PlcTask Outputs/Robot_UR5.UR_inputs/Bits/B17 <-> API/Term 11 (9_O2T General Purpose Registers 1)/Subterm 15 (9_O2T General Purpose Registers 1)/Outputs/O2T Reg 1[2] @bit 1
//     PlcTask Outputs/Robot_UR5.UR_inputs/Bits/B18 <-> API/Term 11 (9_O2T General Purpose Registers 1)/Subterm 15 (9_O2T General Purpose Registers 1)/Outputs/O2T Reg 1[2] @bit 2
//     PlcTask Outputs/Robot_UR5.UR_inputs/Bits/B19 <-> API/Term 11 (9_O2T General Purpose Registers 1)/Subterm 15 (9_O2T General Purpose Registers 1)/Outputs/O2T Reg 1[2] @bit 3
//     PlcTask Outputs/Robot_UR5.UR_inputs/Bits/B2 <-> API/Term 11 (9_O2T General Purpose Registers 1)/Subterm 15 (9_O2T General Purpose Registers 1)/Outputs/O2T Reg 1[0] @bit 2
//     PlcTask Outputs/Robot_UR5.UR_inputs/Bits/B20 <-> API/Term 11 (9_O2T General Purpose Registers 1)/Subterm 15 (9_O2T General Purpose Registers 1)/Outputs/O2T Reg 1[2] @bit 4
//     PlcTask Outputs/Robot_UR5.UR_inputs/Bits/B21 <-> API/Term 11 (9_O2T General Purpose Registers 1)/Subterm 15 (9_O2T General Purpose Registers 1)/Outputs/O2T Reg 1[2] @bit 5
//     PlcTask Outputs/Robot_UR5.UR_inputs/Bits/B22 <-> API/Term 11 (9_O2T General Purpose Registers 1)/Subterm 15 (9_O2T General Purpose Registers 1)/Outputs/O2T Reg 1[2] @bit 6
//     PlcTask Outputs/Robot_UR5.UR_inputs/Bits/B23 <-> API/Term 11 (9_O2T General Purpose Registers 1)/Subterm 15 (9_O2T General Purpose Registers 1)/Outputs/O2T Reg 1[2] @bit 7
//     PlcTask Outputs/Robot_UR5.UR_inputs/Bits/B25 <-> API/Term 11 (9_O2T General Purpose Registers 1)/Subterm 15 (9_O2T General Purpose Registers 1)/Outputs/O2T Reg 1[3] @bit 1
//     PlcTask Outputs/Robot_UR5.UR_inputs/Bits/B26 <-> API/Term 11 (9_O2T General Purpose Registers 1)/Subterm 15 (9_O2T General Purpose Registers 1)/Outputs/O2T Reg 1[3] @bit 2
//     PlcTask Outputs/Robot_UR5.UR_inputs/Bits/B27 <-> API/Term 11 (9_O2T General Purpose Registers 1)/Subterm 15 (9_O2T General Purpose Registers 1)/Outputs/O2T Reg 1[3] @bit 3
//     PlcTask Outputs/Robot_UR5.UR_inputs/Bits/B28 <-> API/Term 11 (9_O2T General Purpose Registers 1)/Subterm 15 (9_O2T General Purpose Registers 1)/Outputs/O2T Reg 1[3] @bit 4
//     PlcTask Outputs/Robot_UR5.UR_inputs/Bits/B29 <-> API/Term 11 (9_O2T General Purpose Registers 1)/Subterm 15 (9_O2T General Purpose Registers 1)/Outputs/O2T Reg 1[3] @bit 5
//     PlcTask Outputs/Robot_UR5.UR_inputs/Bits/B3 <-> API/Term 11 (9_O2T General Purpose Registers 1)/Subterm 15 (9_O2T General Purpose Registers 1)/Outputs/O2T Reg 1[0] @bit 3
//     PlcTask Outputs/Robot_UR5.UR_inputs/Bits/B30 <-> API/Term 11 (9_O2T General Purpose Registers 1)/Subterm 15 (9_O2T General Purpose Registers 1)/Outputs/O2T Reg 1[3] @bit 6
//     PlcTask Outputs/Robot_UR5.UR_inputs/Bits/B31 <-> API/Term 11 (9_O2T General Purpose Registers 1)/Subterm 15 (9_O2T General Purpose Registers 1)/Outputs/O2T Reg 1[3] @bit 7
//     PlcTask Outputs/Robot_UR5.UR_inputs/Bits/B4 <-> API/Term 11 (9_O2T General Purpose Registers 1)/Subterm 15 (9_O2T General Purpose Registers 1)/Outputs/O2T Reg 1[0] @bit 4
//     PlcTask Outputs/Robot_UR5.UR_inputs/Bits/B5 <-> API/Term 11 (9_O2T General Purpose Registers 1)/Subterm 15 (9_O2T General Purpose Registers 1)/Outputs/O2T Reg 1[0] @bit 5
//     PlcTask Outputs/Robot_UR5.UR_inputs/Bits/B6 <-> API/Term 11 (9_O2T General Purpose Registers 1)/Subterm 15 (9_O2T General Purpose Registers 1)/Outputs/O2T Reg 1[0] @bit 6
//     PlcTask Outputs/Robot_UR5.UR_inputs/Bits/B7 <-> API/Term 11 (9_O2T General Purpose Registers 1)/Subterm 15 (9_O2T General Purpose Registers 1)/Outputs/O2T Reg 1[0] @bit 7
//     PlcTask Outputs/Robot_UR5.UR_inputs/Bits/B9 <-> API/Term 11 (9_O2T General Purpose Registers 1)/Subterm 15 (9_O2T General Purpose Registers 1)/Outputs/O2T Reg 1[1] @bit 1
//     PlcTask Outputs/Robot_UR5.UR_inputs/Floats/FLOAT0[0] <-> API/Term 11 (9_O2T General Purpose Registers 1)/Subterm 15 (9_O2T General Purpose Registers 1)/Outputs/O2T Reg 1[52]
//     PlcTask Outputs/Robot_UR5.UR_inputs/Floats/FLOAT0[1] <-> API/Term 11 (9_O2T General Purpose Registers 1)/Subterm 15 (9_O2T General Purpose Registers 1)/Outputs/O2T Reg 1[53]
//     PlcTask Outputs/Robot_UR5.UR_inputs/Floats/FLOAT0[2] <-> API/Term 11 (9_O2T General Purpose Registers 1)/Subterm 15 (9_O2T General Purpose Registers 1)/Outputs/O2T Reg 1[54]
//     PlcTask Outputs/Robot_UR5.UR_inputs/Floats/FLOAT0[3] <-> API/Term 11 (9_O2T General Purpose Registers 1)/Subterm 15 (9_O2T General Purpose Registers 1)/Outputs/O2T Reg 1[55]
//     PlcTask Outputs/Robot_UR5.UR_inputs/Floats/FLOAT10[0] <-> API/Term 11 (9_O2T General Purpose Registers 1)/Subterm 15 (9_O2T General Purpose Registers 1)/Outputs/O2T Reg 1[92]
//     PlcTask Outputs/Robot_UR5.UR_inputs/Floats/FLOAT10[1] <-> API/Term 11 (9_O2T General Purpose Registers 1)/Subterm 15 (9_O2T General Purpose Registers 1)/Outputs/O2T Reg 1[93]
//     PlcTask Outputs/Robot_UR5.UR_inputs/Floats/FLOAT10[2] <-> API/Term 11 (9_O2T General Purpose Registers 1)/Subterm 15 (9_O2T General Purpose Registers 1)/Outputs/O2T Reg 1[94]
//     PlcTask Outputs/Robot_UR5.UR_inputs/Floats/FLOAT10[3] <-> API/Term 11 (9_O2T General Purpose Registers 1)/Subterm 15 (9_O2T General Purpose Registers 1)/Outputs/O2T Reg 1[95]
//     PlcTask Outputs/Robot_UR5.UR_inputs/Floats/FLOAT11[0] <-> API/Term 11 (9_O2T General Purpose Registers 1)/Subterm 15 (9_O2T General Purpose Registers 1)/Outputs/O2T Reg 1[96]
//     PlcTask Outputs/Robot_UR5.UR_inputs/Floats/FLOAT11[1] <-> API/Term 11 (9_O2T General Purpose Registers 1)/Subterm 15 (9_O2T General Purpose Registers 1)/Outputs/O2T Reg 1[97]
//     PlcTask Outputs/Robot_UR5.UR_inputs/Floats/FLOAT11[2] <-> API/Term 11 (9_O2T General Purpose Registers 1)/Subterm 15 (9_O2T General Purpose Registers 1)/Outputs/O2T Reg 1[98]
//     PlcTask Outputs/Robot_UR5.UR_inputs/Floats/FLOAT11[3] <-> API/Term 11 (9_O2T General Purpose Registers 1)/Subterm 15 (9_O2T General Purpose Registers 1)/Outputs/O2T Reg 1[99]
//     PlcTask Outputs/Robot_UR5.UR_inputs/Floats/FLOAT1[0] <-> API/Term 11 (9_O2T General Purpose Registers 1)/Subterm 15 (9_O2T General Purpose Registers 1)/Outputs/O2T Reg 1[56]
//     PlcTask Outputs/Robot_UR5.UR_inputs/Floats/FLOAT1[1] <-> API/Term 11 (9_O2T General Purpose Registers 1)/Subterm 15 (9_O2T General Purpose Registers 1)/Outputs/O2T Reg 1[57]
//     PlcTask Outputs/Robot_UR5.UR_inputs/Floats/FLOAT1[2] <-> API/Term 11 (9_O2T General Purpose Registers 1)/Subterm 15 (9_O2T General Purpose Registers 1)/Outputs/O2T Reg 1[58]
//     PlcTask Outputs/Robot_UR5.UR_inputs/Floats/FLOAT1[3] <-> API/Term 11 (9_O2T General Purpose Registers 1)/Subterm 15 (9_O2T General Purpose Registers 1)/Outputs/O2T Reg 1[59]
//     PlcTask Outputs/Robot_UR5.UR_inputs/Floats/FLOAT2[0] <-> API/Term 11 (9_O2T General Purpose Registers 1)/Subterm 15 (9_O2T General Purpose Registers 1)/Outputs/O2T Reg 1[60]
//     PlcTask Outputs/Robot_UR5.UR_inputs/Floats/FLOAT2[1] <-> API/Term 11 (9_O2T General Purpose Registers 1)/Subterm 15 (9_O2T General Purpose Registers 1)/Outputs/O2T Reg 1[61]
//     PlcTask Outputs/Robot_UR5.UR_inputs/Floats/FLOAT2[2] <-> API/Term 11 (9_O2T General Purpose Registers 1)/Subterm 15 (9_O2T General Purpose Registers 1)/Outputs/O2T Reg 1[62]
//     PlcTask Outputs/Robot_UR5.UR_inputs/Floats/FLOAT2[3] <-> API/Term 11 (9_O2T General Purpose Registers 1)/Subterm 15 (9_O2T General Purpose Registers 1)/Outputs/O2T Reg 1[63]
//     PlcTask Outputs/Robot_UR5.UR_inputs/Floats/FLOAT3[0] <-> API/Term 11 (9_O2T General Purpose Registers 1)/Subterm 15 (9_O2T General Purpose Registers 1)/Outputs/O2T Reg 1[64]
//     PlcTask Outputs/Robot_UR5.UR_inputs/Floats/FLOAT3[1] <-> API/Term 11 (9_O2T General Purpose Registers 1)/Subterm 15 (9_O2T General Purpose Registers 1)/Outputs/O2T Reg 1[65]
//     PlcTask Outputs/Robot_UR5.UR_inputs/Floats/FLOAT3[2] <-> API/Term 11 (9_O2T General Purpose Registers 1)/Subterm 15 (9_O2T General Purpose Registers 1)/Outputs/O2T Reg 1[66]
//     PlcTask Outputs/Robot_UR5.UR_inputs/Floats/FLOAT3[3] <-> API/Term 11 (9_O2T General Purpose Registers 1)/Subterm 15 (9_O2T General Purpose Registers 1)/Outputs/O2T Reg 1[67]
//     PlcTask Outputs/Robot_UR5.UR_inputs/Floats/FLOAT4[0] <-> API/Term 11 (9_O2T General Purpose Registers 1)/Subterm 15 (9_O2T General Purpose Registers 1)/Outputs/O2T Reg 1[68]
//     PlcTask Outputs/Robot_UR5.UR_inputs/Floats/FLOAT4[1] <-> API/Term 11 (9_O2T General Purpose Registers 1)/Subterm 15 (9_O2T General Purpose Registers 1)/Outputs/O2T Reg 1[69]
//     PlcTask Outputs/Robot_UR5.UR_inputs/Floats/FLOAT4[2] <-> API/Term 11 (9_O2T General Purpose Registers 1)/Subterm 15 (9_O2T General Purpose Registers 1)/Outputs/O2T Reg 1[70]
//     PlcTask Outputs/Robot_UR5.UR_inputs/Floats/FLOAT4[3] <-> API/Term 11 (9_O2T General Purpose Registers 1)/Subterm 15 (9_O2T General Purpose Registers 1)/Outputs/O2T Reg 1[71]
//     PlcTask Outputs/Robot_UR5.UR_inputs/Floats/FLOAT5[0] <-> API/Term 11 (9_O2T General Purpose Registers 1)/Subterm 15 (9_O2T General Purpose Registers 1)/Outputs/O2T Reg 1[72]
//     PlcTask Outputs/Robot_UR5.UR_inputs/Floats/FLOAT5[1] <-> API/Term 11 (9_O2T General Purpose Registers 1)/Subterm 15 (9_O2T General Purpose Registers 1)/Outputs/O2T Reg 1[73]
//     PlcTask Outputs/Robot_UR5.UR_inputs/Floats/FLOAT5[2] <-> API/Term 11 (9_O2T General Purpose Registers 1)/Subterm 15 (9_O2T General Purpose Registers 1)/Outputs/O2T Reg 1[74]
//     PlcTask Outputs/Robot_UR5.UR_inputs/Floats/FLOAT5[3] <-> API/Term 11 (9_O2T General Purpose Registers 1)/Subterm 15 (9_O2T General Purpose Registers 1)/Outputs/O2T Reg 1[75]
//     PlcTask Outputs/Robot_UR5.UR_inputs/Floats/FLOAT6[0] <-> API/Term 11 (9_O2T General Purpose Registers 1)/Subterm 15 (9_O2T General Purpose Registers 1)/Outputs/O2T Reg 1[76]
//     PlcTask Outputs/Robot_UR5.UR_inputs/Floats/FLOAT6[1] <-> API/Term 11 (9_O2T General Purpose Registers 1)/Subterm 15 (9_O2T General Purpose Registers 1)/Outputs/O2T Reg 1[77]
//     PlcTask Outputs/Robot_UR5.UR_inputs/Floats/FLOAT6[2] <-> API/Term 11 (9_O2T General Purpose Registers 1)/Subterm 15 (9_O2T General Purpose Registers 1)/Outputs/O2T Reg 1[78]
//     PlcTask Outputs/Robot_UR5.UR_inputs/Floats/FLOAT6[3] <-> API/Term 11 (9_O2T General Purpose Registers 1)/Subterm 15 (9_O2T General Purpose Registers 1)/Outputs/O2T Reg 1[79]
//     PlcTask Outputs/Robot_UR5.UR_inputs/Floats/FLOAT7[0] <-> API/Term 11 (9_O2T General Purpose Registers 1)/Subterm 15 (9_O2T General Purpose Registers 1)/Outputs/O2T Reg 1[80]
//     PlcTask Outputs/Robot_UR5.UR_inputs/Floats/FLOAT7[1] <-> API/Term 11 (9_O2T General Purpose Registers 1)/Subterm 15 (9_O2T General Purpose Registers 1)/Outputs/O2T Reg 1[81]
//     PlcTask Outputs/Robot_UR5.UR_inputs/Floats/FLOAT7[2] <-> API/Term 11 (9_O2T General Purpose Registers 1)/Subterm 15 (9_O2T General Purpose Registers 1)/Outputs/O2T Reg 1[82]
//     PlcTask Outputs/Robot_UR5.UR_inputs/Floats/FLOAT7[3] <-> API/Term 11 (9_O2T General Purpose Registers 1)/Subterm 15 (9_O2T General Purpose Registers 1)/Outputs/O2T Reg 1[83]
//     PlcTask Outputs/Robot_UR5.UR_inputs/Floats/FLOAT8[0] <-> API/Term 11 (9_O2T General Purpose Registers 1)/Subterm 15 (9_O2T General Purpose Registers 1)/Outputs/O2T Reg 1[84]
//     PlcTask Outputs/Robot_UR5.UR_inputs/Floats/FLOAT8[1] <-> API/Term 11 (9_O2T General Purpose Registers 1)/Subterm 15 (9_O2T General Purpose Registers 1)/Outputs/O2T Reg 1[85]
//     PlcTask Outputs/Robot_UR5.UR_inputs/Floats/FLOAT8[2] <-> API/Term 11 (9_O2T General Purpose Registers 1)/Subterm 15 (9_O2T General Purpose Registers 1)/Outputs/O2T Reg 1[86]
//     PlcTask Outputs/Robot_UR5.UR_inputs/Floats/FLOAT8[3] <-> API/Term 11 (9_O2T General Purpose Registers 1)/Subterm 15 (9_O2T General Purpose Registers 1)/Outputs/O2T Reg 1[87]
//     PlcTask Outputs/Robot_UR5.UR_inputs/Floats/FLOAT9[0] <-> API/Term 11 (9_O2T General Purpose Registers 1)/Subterm 15 (9_O2T General Purpose Registers 1)/Outputs/O2T Reg 1[88]
//     PlcTask Outputs/Robot_UR5.UR_inputs/Floats/FLOAT9[1] <-> API/Term 11 (9_O2T General Purpose Registers 1)/Subterm 15 (9_O2T General Purpose Registers 1)/Outputs/O2T Reg 1[89]
//     PlcTask Outputs/Robot_UR5.UR_inputs/Floats/FLOAT9[2] <-> API/Term 11 (9_O2T General Purpose Registers 1)/Subterm 15 (9_O2T General Purpose Registers 1)/Outputs/O2T Reg 1[90]
//     PlcTask Outputs/Robot_UR5.UR_inputs/Floats/FLOAT9[3] <-> API/Term 11 (9_O2T General Purpose Registers 1)/Subterm 15 (9_O2T General Purpose Registers 1)/Outputs/O2T Reg 1[91]
//     PlcTask Outputs/Robot_UR5.UR_inputs/Ints/INT0[0] <-> API/Term 11 (9_O2T General Purpose Registers 1)/Subterm 15 (9_O2T General Purpose Registers 1)/Outputs/O2T Reg 1[4]
//     PlcTask Outputs/Robot_UR5.UR_inputs/Ints/INT0[1] <-> API/Term 11 (9_O2T General Purpose Registers 1)/Subterm 15 (9_O2T General Purpose Registers 1)/Outputs/O2T Reg 1[5]
//     PlcTask Outputs/Robot_UR5.UR_inputs/Ints/INT0[2] <-> API/Term 11 (9_O2T General Purpose Registers 1)/Subterm 15 (9_O2T General Purpose Registers 1)/Outputs/O2T Reg 1[6]
//     PlcTask Outputs/Robot_UR5.UR_inputs/Ints/INT0[3] <-> API/Term 11 (9_O2T General Purpose Registers 1)/Subterm 15 (9_O2T General Purpose Registers 1)/Outputs/O2T Reg 1[7]
//     PlcTask Outputs/Robot_UR5.UR_inputs/Ints/INT10[0] <-> API/Term 11 (9_O2T General Purpose Registers 1)/Subterm 15 (9_O2T General Purpose Registers 1)/Outputs/O2T Reg 1[44]
//     PlcTask Outputs/Robot_UR5.UR_inputs/Ints/INT10[1] <-> API/Term 11 (9_O2T General Purpose Registers 1)/Subterm 15 (9_O2T General Purpose Registers 1)/Outputs/O2T Reg 1[45]
//     PlcTask Outputs/Robot_UR5.UR_inputs/Ints/INT10[2] <-> API/Term 11 (9_O2T General Purpose Registers 1)/Subterm 15 (9_O2T General Purpose Registers 1)/Outputs/O2T Reg 1[46]
//     PlcTask Outputs/Robot_UR5.UR_inputs/Ints/INT10[3] <-> API/Term 11 (9_O2T General Purpose Registers 1)/Subterm 15 (9_O2T General Purpose Registers 1)/Outputs/O2T Reg 1[47]
//     PlcTask Outputs/Robot_UR5.UR_inputs/Ints/INT11[0] <-> API/Term 11 (9_O2T General Purpose Registers 1)/Subterm 15 (9_O2T General Purpose Registers 1)/Outputs/O2T Reg 1[48]
//     PlcTask Outputs/Robot_UR5.UR_inputs/Ints/INT11[1] <-> API/Term 11 (9_O2T General Purpose Registers 1)/Subterm 15 (9_O2T General Purpose Registers 1)/Outputs/O2T Reg 1[49]
//     PlcTask Outputs/Robot_UR5.UR_inputs/Ints/INT11[2] <-> API/Term 11 (9_O2T General Purpose Registers 1)/Subterm 15 (9_O2T General Purpose Registers 1)/Outputs/O2T Reg 1[50]
//     PlcTask Outputs/Robot_UR5.UR_inputs/Ints/INT11[3] <-> API/Term 11 (9_O2T General Purpose Registers 1)/Subterm 15 (9_O2T General Purpose Registers 1)/Outputs/O2T Reg 1[51]
//     PlcTask Outputs/Robot_UR5.UR_inputs/Ints/INT1[0] <-> API/Term 11 (9_O2T General Purpose Registers 1)/Subterm 15 (9_O2T General Purpose Registers 1)/Outputs/O2T Reg 1[8]
//     PlcTask Outputs/Robot_UR5.UR_inputs/Ints/INT1[1] <-> API/Term 11 (9_O2T General Purpose Registers 1)/Subterm 15 (9_O2T General Purpose Registers 1)/Outputs/O2T Reg 1[9]
//     PlcTask Outputs/Robot_UR5.UR_inputs/Ints/INT1[2] <-> API/Term 11 (9_O2T General Purpose Registers 1)/Subterm 15 (9_O2T General Purpose Registers 1)/Outputs/O2T Reg 1[10]
//     PlcTask Outputs/Robot_UR5.UR_inputs/Ints/INT1[3] <-> API/Term 11 (9_O2T General Purpose Registers 1)/Subterm 15 (9_O2T General Purpose Registers 1)/Outputs/O2T Reg 1[11]
//     PlcTask Outputs/Robot_UR5.UR_inputs/Ints/INT2[0] <-> API/Term 11 (9_O2T General Purpose Registers 1)/Subterm 15 (9_O2T General Purpose Registers 1)/Outputs/O2T Reg 1[12]
//     PlcTask Outputs/Robot_UR5.UR_inputs/Ints/INT2[1] <-> API/Term 11 (9_O2T General Purpose Registers 1)/Subterm 15 (9_O2T General Purpose Registers 1)/Outputs/O2T Reg 1[13]
//     PlcTask Outputs/Robot_UR5.UR_inputs/Ints/INT2[2] <-> API/Term 11 (9_O2T General Purpose Registers 1)/Subterm 15 (9_O2T General Purpose Registers 1)/Outputs/O2T Reg 1[14]
//     PlcTask Outputs/Robot_UR5.UR_inputs/Ints/INT2[3] <-> API/Term 11 (9_O2T General Purpose Registers 1)/Subterm 15 (9_O2T General Purpose Registers 1)/Outputs/O2T Reg 1[15]
//     PlcTask Outputs/Robot_UR5.UR_inputs/Ints/INT3[0] <-> API/Term 11 (9_O2T General Purpose Registers 1)/Subterm 15 (9_O2T General Purpose Registers 1)/Outputs/O2T Reg 1[16]
//     PlcTask Outputs/Robot_UR5.UR_inputs/Ints/INT3[1] <-> API/Term 11 (9_O2T General Purpose Registers 1)/Subterm 15 (9_O2T General Purpose Registers 1)/Outputs/O2T Reg 1[17]
//     PlcTask Outputs/Robot_UR5.UR_inputs/Ints/INT3[2] <-> API/Term 11 (9_O2T General Purpose Registers 1)/Subterm 15 (9_O2T General Purpose Registers 1)/Outputs/O2T Reg 1[18]
//     PlcTask Outputs/Robot_UR5.UR_inputs/Ints/INT3[3] <-> API/Term 11 (9_O2T General Purpose Registers 1)/Subterm 15 (9_O2T General Purpose Registers 1)/Outputs/O2T Reg 1[19]
//     PlcTask Outputs/Robot_UR5.UR_inputs/Ints/INT4[0] <-> API/Term 11 (9_O2T General Purpose Registers 1)/Subterm 15 (9_O2T General Purpose Registers 1)/Outputs/O2T Reg 1[20]
//     PlcTask Outputs/Robot_UR5.UR_inputs/Ints/INT4[1] <-> API/Term 11 (9_O2T General Purpose Registers 1)/Subterm 15 (9_O2T General Purpose Registers 1)/Outputs/O2T Reg 1[21]
//     PlcTask Outputs/Robot_UR5.UR_inputs/Ints/INT4[2] <-> API/Term 11 (9_O2T General Purpose Registers 1)/Subterm 15 (9_O2T General Purpose Registers 1)/Outputs/O2T Reg 1[22]
//     PlcTask Outputs/Robot_UR5.UR_inputs/Ints/INT4[3] <-> API/Term 11 (9_O2T General Purpose Registers 1)/Subterm 15 (9_O2T General Purpose Registers 1)/Outputs/O2T Reg 1[23]
//     PlcTask Outputs/Robot_UR5.UR_inputs/Ints/INT5[0] <-> API/Term 11 (9_O2T General Purpose Registers 1)/Subterm 15 (9_O2T General Purpose Registers 1)/Outputs/O2T Reg 1[24]
//     PlcTask Outputs/Robot_UR5.UR_inputs/Ints/INT5[1] <-> API/Term 11 (9_O2T General Purpose Registers 1)/Subterm 15 (9_O2T General Purpose Registers 1)/Outputs/O2T Reg 1[25]
//     PlcTask Outputs/Robot_UR5.UR_inputs/Ints/INT5[2] <-> API/Term 11 (9_O2T General Purpose Registers 1)/Subterm 15 (9_O2T General Purpose Registers 1)/Outputs/O2T Reg 1[26]
//     PlcTask Outputs/Robot_UR5.UR_inputs/Ints/INT5[3] <-> API/Term 11 (9_O2T General Purpose Registers 1)/Subterm 15 (9_O2T General Purpose Registers 1)/Outputs/O2T Reg 1[27]
//     PlcTask Outputs/Robot_UR5.UR_inputs/Ints/INT6[0] <-> API/Term 11 (9_O2T General Purpose Registers 1)/Subterm 15 (9_O2T General Purpose Registers 1)/Outputs/O2T Reg 1[28]
//     PlcTask Outputs/Robot_UR5.UR_inputs/Ints/INT6[1] <-> API/Term 11 (9_O2T General Purpose Registers 1)/Subterm 15 (9_O2T General Purpose Registers 1)/Outputs/O2T Reg 1[29]
//     PlcTask Outputs/Robot_UR5.UR_inputs/Ints/INT6[2] <-> API/Term 11 (9_O2T General Purpose Registers 1)/Subterm 15 (9_O2T General Purpose Registers 1)/Outputs/O2T Reg 1[30]
//     PlcTask Outputs/Robot_UR5.UR_inputs/Ints/INT6[3] <-> API/Term 11 (9_O2T General Purpose Registers 1)/Subterm 15 (9_O2T General Purpose Registers 1)/Outputs/O2T Reg 1[31]
//     PlcTask Outputs/Robot_UR5.UR_inputs/Ints/INT7[0] <-> API/Term 11 (9_O2T General Purpose Registers 1)/Subterm 15 (9_O2T General Purpose Registers 1)/Outputs/O2T Reg 1[32]
//     PlcTask Outputs/Robot_UR5.UR_inputs/Ints/INT7[1] <-> API/Term 11 (9_O2T General Purpose Registers 1)/Subterm 15 (9_O2T General Purpose Registers 1)/Outputs/O2T Reg 1[33]
//     PlcTask Outputs/Robot_UR5.UR_inputs/Ints/INT7[2] <-> API/Term 11 (9_O2T General Purpose Registers 1)/Subterm 15 (9_O2T General Purpose Registers 1)/Outputs/O2T Reg 1[34]
//     PlcTask Outputs/Robot_UR5.UR_inputs/Ints/INT7[3] <-> API/Term 11 (9_O2T General Purpose Registers 1)/Subterm 15 (9_O2T General Purpose Registers 1)/Outputs/O2T Reg 1[35]
//     PlcTask Outputs/Robot_UR5.UR_inputs/Ints/INT8[0] <-> API/Term 11 (9_O2T General Purpose Registers 1)/Subterm 15 (9_O2T General Purpose Registers 1)/Outputs/O2T Reg 1[36]
//     PlcTask Outputs/Robot_UR5.UR_inputs/Ints/INT8[1] <-> API/Term 11 (9_O2T General Purpose Registers 1)/Subterm 15 (9_O2T General Purpose Registers 1)/Outputs/O2T Reg 1[37]
//     PlcTask Outputs/Robot_UR5.UR_inputs/Ints/INT8[2] <-> API/Term 11 (9_O2T General Purpose Registers 1)/Subterm 15 (9_O2T General Purpose Registers 1)/Outputs/O2T Reg 1[38]
//     PlcTask Outputs/Robot_UR5.UR_inputs/Ints/INT8[3] <-> API/Term 11 (9_O2T General Purpose Registers 1)/Subterm 15 (9_O2T General Purpose Registers 1)/Outputs/O2T Reg 1[39]
//     PlcTask Outputs/Robot_UR5.UR_inputs/Ints/INT9[0] <-> API/Term 11 (9_O2T General Purpose Registers 1)/Subterm 15 (9_O2T General Purpose Registers 1)/Outputs/O2T Reg 1[40]
//     PlcTask Outputs/Robot_UR5.UR_inputs/Ints/INT9[1] <-> API/Term 11 (9_O2T General Purpose Registers 1)/Subterm 15 (9_O2T General Purpose Registers 1)/Outputs/O2T Reg 1[41]
//     PlcTask Outputs/Robot_UR5.UR_inputs/Ints/INT9[2] <-> API/Term 11 (9_O2T General Purpose Registers 1)/Subterm 15 (9_O2T General Purpose Registers 1)/Outputs/O2T Reg 1[42]
//     PlcTask Outputs/Robot_UR5.UR_inputs/Ints/INT9[3] <-> API/Term 11 (9_O2T General Purpose Registers 1)/Subterm 15 (9_O2T General Purpose Registers 1)/Outputs/O2T Reg 1[43]
//     PlcTask Outputs/Robot_UR5.UR_inputs_2/Floats/FLOAT12[0] <-> API/Term 12 (10_O2T General Purpose Registers 2)/Subterm 16 (10_O2T General Purpose Registers 2)/Outputs/O2T Reg 2[52]
//     PlcTask Outputs/Robot_UR5.UR_inputs_2/Floats/FLOAT12[1] <-> API/Term 12 (10_O2T General Purpose Registers 2)/Subterm 16 (10_O2T General Purpose Registers 2)/Outputs/O2T Reg 2[53]
//     PlcTask Outputs/Robot_UR5.UR_inputs_2/Floats/FLOAT12[2] <-> API/Term 12 (10_O2T General Purpose Registers 2)/Subterm 16 (10_O2T General Purpose Registers 2)/Outputs/O2T Reg 2[54]
//     PlcTask Outputs/Robot_UR5.UR_inputs_2/Floats/FLOAT12[3] <-> API/Term 12 (10_O2T General Purpose Registers 2)/Subterm 16 (10_O2T General Purpose Registers 2)/Outputs/O2T Reg 2[55]
//     PlcTask Outputs/Robot_UR5.UR_inputs_2/Floats/FLOAT13[0] <-> API/Term 12 (10_O2T General Purpose Registers 2)/Subterm 16 (10_O2T General Purpose Registers 2)/Outputs/O2T Reg 2[56]
//     PlcTask Outputs/Robot_UR5.UR_inputs_2/Floats/FLOAT13[1] <-> API/Term 12 (10_O2T General Purpose Registers 2)/Subterm 16 (10_O2T General Purpose Registers 2)/Outputs/O2T Reg 2[57]
//     PlcTask Outputs/Robot_UR5.UR_inputs_2/Floats/FLOAT13[2] <-> API/Term 12 (10_O2T General Purpose Registers 2)/Subterm 16 (10_O2T General Purpose Registers 2)/Outputs/O2T Reg 2[58]
//     PlcTask Outputs/Robot_UR5.UR_inputs_2/Floats/FLOAT13[3] <-> API/Term 12 (10_O2T General Purpose Registers 2)/Subterm 16 (10_O2T General Purpose Registers 2)/Outputs/O2T Reg 2[59]
//     PlcTask Outputs/Robot_UR5.UR_inputs_2/Floats/FLOAT14[0] <-> API/Term 12 (10_O2T General Purpose Registers 2)/Subterm 16 (10_O2T General Purpose Registers 2)/Outputs/O2T Reg 2[60]
//     PlcTask Outputs/Robot_UR5.UR_inputs_2/Floats/FLOAT14[1] <-> API/Term 12 (10_O2T General Purpose Registers 2)/Subterm 16 (10_O2T General Purpose Registers 2)/Outputs/O2T Reg 2[61]
//     PlcTask Outputs/Robot_UR5.UR_inputs_2/Floats/FLOAT14[2] <-> API/Term 12 (10_O2T General Purpose Registers 2)/Subterm 16 (10_O2T General Purpose Registers 2)/Outputs/O2T Reg 2[62]
//     PlcTask Outputs/Robot_UR5.UR_inputs_2/Floats/FLOAT14[3] <-> API/Term 12 (10_O2T General Purpose Registers 2)/Subterm 16 (10_O2T General Purpose Registers 2)/Outputs/O2T Reg 2[63]
//     PlcTask Outputs/Robot_UR5.UR_inputs_2/Floats/FLOAT15[0] <-> API/Term 12 (10_O2T General Purpose Registers 2)/Subterm 16 (10_O2T General Purpose Registers 2)/Outputs/O2T Reg 2[64]
//     PlcTask Outputs/Robot_UR5.UR_inputs_2/Floats/FLOAT15[1] <-> API/Term 12 (10_O2T General Purpose Registers 2)/Subterm 16 (10_O2T General Purpose Registers 2)/Outputs/O2T Reg 2[65]
//     PlcTask Outputs/Robot_UR5.UR_inputs_2/Floats/FLOAT15[2] <-> API/Term 12 (10_O2T General Purpose Registers 2)/Subterm 16 (10_O2T General Purpose Registers 2)/Outputs/O2T Reg 2[66]
//     PlcTask Outputs/Robot_UR5.UR_inputs_2/Floats/FLOAT15[3] <-> API/Term 12 (10_O2T General Purpose Registers 2)/Subterm 16 (10_O2T General Purpose Registers 2)/Outputs/O2T Reg 2[67]
//     PlcTask Outputs/Robot_UR5.UR_inputs_2/Floats/FLOAT16[0] <-> API/Term 12 (10_O2T General Purpose Registers 2)/Subterm 16 (10_O2T General Purpose Registers 2)/Outputs/O2T Reg 2[68]
//     PlcTask Outputs/Robot_UR5.UR_inputs_2/Floats/FLOAT16[1] <-> API/Term 12 (10_O2T General Purpose Registers 2)/Subterm 16 (10_O2T General Purpose Registers 2)/Outputs/O2T Reg 2[69]
//     PlcTask Outputs/Robot_UR5.UR_inputs_2/Floats/FLOAT16[2] <-> API/Term 12 (10_O2T General Purpose Registers 2)/Subterm 16 (10_O2T General Purpose Registers 2)/Outputs/O2T Reg 2[70]
//     PlcTask Outputs/Robot_UR5.UR_inputs_2/Floats/FLOAT16[3] <-> API/Term 12 (10_O2T General Purpose Registers 2)/Subterm 16 (10_O2T General Purpose Registers 2)/Outputs/O2T Reg 2[71]
//     PlcTask Outputs/Robot_UR5.UR_inputs_2/Floats/FLOAT17[0] <-> API/Term 12 (10_O2T General Purpose Registers 2)/Subterm 16 (10_O2T General Purpose Registers 2)/Outputs/O2T Reg 2[72]
//     PlcTask Outputs/Robot_UR5.UR_inputs_2/Floats/FLOAT17[1] <-> API/Term 12 (10_O2T General Purpose Registers 2)/Subterm 16 (10_O2T General Purpose Registers 2)/Outputs/O2T Reg 2[73]
//     PlcTask Outputs/Robot_UR5.UR_inputs_2/Floats/FLOAT17[2] <-> API/Term 12 (10_O2T General Purpose Registers 2)/Subterm 16 (10_O2T General Purpose Registers 2)/Outputs/O2T Reg 2[74]
//     PlcTask Outputs/Robot_UR5.UR_inputs_2/Floats/FLOAT17[3] <-> API/Term 12 (10_O2T General Purpose Registers 2)/Subterm 16 (10_O2T General Purpose Registers 2)/Outputs/O2T Reg 2[75]
//     PlcTask Outputs/Robot_UR5.UR_inputs_2/Floats/FLOAT18[0] <-> API/Term 12 (10_O2T General Purpose Registers 2)/Subterm 16 (10_O2T General Purpose Registers 2)/Outputs/O2T Reg 2[76]
//     PlcTask Outputs/Robot_UR5.UR_inputs_2/Floats/FLOAT18[1] <-> API/Term 12 (10_O2T General Purpose Registers 2)/Subterm 16 (10_O2T General Purpose Registers 2)/Outputs/O2T Reg 2[77]
//     PlcTask Outputs/Robot_UR5.UR_inputs_2/Floats/FLOAT18[2] <-> API/Term 12 (10_O2T General Purpose Registers 2)/Subterm 16 (10_O2T General Purpose Registers 2)/Outputs/O2T Reg 2[78]
//     PlcTask Outputs/Robot_UR5.UR_inputs_2/Floats/FLOAT18[3] <-> API/Term 12 (10_O2T General Purpose Registers 2)/Subterm 16 (10_O2T General Purpose Registers 2)/Outputs/O2T Reg 2[79]
//     PlcTask Outputs/Robot_UR5.UR_inputs_2/Floats/FLOAT19[0] <-> API/Term 12 (10_O2T General Purpose Registers 2)/Subterm 16 (10_O2T General Purpose Registers 2)/Outputs/O2T Reg 2[80]
//     PlcTask Outputs/Robot_UR5.UR_inputs_2/Floats/FLOAT19[1] <-> API/Term 12 (10_O2T General Purpose Registers 2)/Subterm 16 (10_O2T General Purpose Registers 2)/Outputs/O2T Reg 2[81]
//     PlcTask Outputs/Robot_UR5.UR_inputs_2/Floats/FLOAT19[2] <-> API/Term 12 (10_O2T General Purpose Registers 2)/Subterm 16 (10_O2T General Purpose Registers 2)/Outputs/O2T Reg 2[82]
//     PlcTask Outputs/Robot_UR5.UR_inputs_2/Floats/FLOAT19[3] <-> API/Term 12 (10_O2T General Purpose Registers 2)/Subterm 16 (10_O2T General Purpose Registers 2)/Outputs/O2T Reg 2[83]
//     PlcTask Outputs/Robot_UR5.UR_inputs_2/Floats/FLOAT20[0] <-> API/Term 12 (10_O2T General Purpose Registers 2)/Subterm 16 (10_O2T General Purpose Registers 2)/Outputs/O2T Reg 2[84]
//     PlcTask Outputs/Robot_UR5.UR_inputs_2/Floats/FLOAT20[1] <-> API/Term 12 (10_O2T General Purpose Registers 2)/Subterm 16 (10_O2T General Purpose Registers 2)/Outputs/O2T Reg 2[85]
//     PlcTask Outputs/Robot_UR5.UR_inputs_2/Floats/FLOAT20[2] <-> API/Term 12 (10_O2T General Purpose Registers 2)/Subterm 16 (10_O2T General Purpose Registers 2)/Outputs/O2T Reg 2[86]
//     PlcTask Outputs/Robot_UR5.UR_inputs_2/Floats/FLOAT20[3] <-> API/Term 12 (10_O2T General Purpose Registers 2)/Subterm 16 (10_O2T General Purpose Registers 2)/Outputs/O2T Reg 2[87]
//     PlcTask Outputs/Robot_UR5.UR_inputs_2/Floats/FLOAT21[0] <-> API/Term 12 (10_O2T General Purpose Registers 2)/Subterm 16 (10_O2T General Purpose Registers 2)/Outputs/O2T Reg 2[88]
//     PlcTask Outputs/Robot_UR5.UR_inputs_2/Floats/FLOAT21[1] <-> API/Term 12 (10_O2T General Purpose Registers 2)/Subterm 16 (10_O2T General Purpose Registers 2)/Outputs/O2T Reg 2[89]
//     PlcTask Outputs/Robot_UR5.UR_inputs_2/Floats/FLOAT21[2] <-> API/Term 12 (10_O2T General Purpose Registers 2)/Subterm 16 (10_O2T General Purpose Registers 2)/Outputs/O2T Reg 2[90]
//     PlcTask Outputs/Robot_UR5.UR_inputs_2/Floats/FLOAT21[3] <-> API/Term 12 (10_O2T General Purpose Registers 2)/Subterm 16 (10_O2T General Purpose Registers 2)/Outputs/O2T Reg 2[91]
//     PlcTask Outputs/Robot_UR5.UR_inputs_2/Floats/FLOAT22[0] <-> API/Term 12 (10_O2T General Purpose Registers 2)/Subterm 16 (10_O2T General Purpose Registers 2)/Outputs/O2T Reg 2[92]
//     PlcTask Outputs/Robot_UR5.UR_inputs_2/Floats/FLOAT22[1] <-> API/Term 12 (10_O2T General Purpose Registers 2)/Subterm 16 (10_O2T General Purpose Registers 2)/Outputs/O2T Reg 2[93]
//     PlcTask Outputs/Robot_UR5.UR_inputs_2/Floats/FLOAT22[2] <-> API/Term 12 (10_O2T General Purpose Registers 2)/Subterm 16 (10_O2T General Purpose Registers 2)/Outputs/O2T Reg 2[94]
//     PlcTask Outputs/Robot_UR5.UR_inputs_2/Floats/FLOAT22[3] <-> API/Term 12 (10_O2T General Purpose Registers 2)/Subterm 16 (10_O2T General Purpose Registers 2)/Outputs/O2T Reg 2[95]
//     PlcTask Outputs/Robot_UR5.UR_inputs_2/Floats/FLOAT23[0] <-> API/Term 12 (10_O2T General Purpose Registers 2)/Subterm 16 (10_O2T General Purpose Registers 2)/Outputs/O2T Reg 2[96]
//     PlcTask Outputs/Robot_UR5.UR_inputs_2/Floats/FLOAT23[1] <-> API/Term 12 (10_O2T General Purpose Registers 2)/Subterm 16 (10_O2T General Purpose Registers 2)/Outputs/O2T Reg 2[97]
//     PlcTask Outputs/Robot_UR5.UR_inputs_2/Floats/FLOAT23[2] <-> API/Term 12 (10_O2T General Purpose Registers 2)/Subterm 16 (10_O2T General Purpose Registers 2)/Outputs/O2T Reg 2[98]
//     PlcTask Outputs/Robot_UR5.UR_inputs_2/Floats/FLOAT23[3] <-> API/Term 12 (10_O2T General Purpose Registers 2)/Subterm 16 (10_O2T General Purpose Registers 2)/Outputs/O2T Reg 2[99]
//   p1/p1 Instance <-> Device 5 (EtherCAT)/Drive 1 (ZeroErr Driver)
//     PlcTask Inputs/QRob_StateMachine.Qrob_torque <-> Transmit PDO mapping 0/Current Actual Value
//     PlcTask Inputs/QRob_StateMachine.Qrob_velocity <-> Transmit PDO mapping 0/Actual velocity
//   p1/p1 Instance <-> Device 7 (EtherCAT)/Term 4 (EK1100)/Term 12 (EL1809)
//     PlcTask Inputs/QRob_StateMachine.Sensor_Position_detection <-> Channel 16/Input
//   p1/p1 Instance <-> Device 7 (EtherCAT)/Term 4 (EK1100)/Term 5 (EL2809)
//     PlcTask Outputs/Get_QRob_Pos.Cooler_fan <-> Channel 9/Output
//     PlcTask Outputs/UR3_StateMachine.UR3_Power_on <-> Channel 8/Output
//     PlcTask Outputs/UR5_StateMachine.UR5_Power_on <-> Channel 4/Output
//     PlcTask Outputs/UR3_StateMachine.UR3_Run_Robot <-> Channel 7/Output
//     PlcTask Outputs/UR5_StateMachine.UR5_Run_Robot <-> Channel 3/Output
//     PlcTask Outputs/UR3_StateMachine.UR3_Safety_pin_1 <-> Channel 5/Output
//     PlcTask Outputs/UR3_StateMachine.UR3_Safety_pin_2 <-> Channel 6/Output
//     PlcTask Outputs/UR5_StateMachine.UR5_Safety_pin_1 <-> Channel 1/Output
//     PlcTask Outputs/UR5_StateMachine.UR5_Safety_pin_2 <-> Channel 2/Output
//   p1/p1 Instance <-> NC-Task 1 SAF/Axes/Axis 1
//     PlcTask Inputs/Global_Servo.Axis1.NcToPlc <-> Outputs/ToPlc
//     PlcTask Outputs/Global_Servo.Axis1.PlcToNc <-> Inputs/FromPlc

CONFIGURATION p1
    RESOURCE PLC ON TwinCAT3
        TASK PlcTask(INTERVAL := T#1ms, PRIORITY := 4);
        PROGRAM MASTER_CTR WITH PlcTask : MASTER_CTR;
        PROGRAM QRob_StateMachine WITH PlcTask : QRob_StateMachine;
        PROGRAM Get_QRob_Pos WITH PlcTask : Get_QRob_Pos;
        PROGRAM UR5_StateMachine WITH PlcTask : UR5_StateMachine;
        PROGRAM UR3_StateMachine WITH PlcTask : UR3_StateMachine;
        PROGRAM Vision_StateMachine WITH PlcTask : Vision_StateMachine;
    END_RESOURCE
END_CONFIGURATION

// ---- DUTs/UR_10 _O2T_Registers/UR_10_O2T_Registers.TcDUT
TYPE UR_10_O2T_Registers :
STRUCT
	  Bits : UR_O2T_bits_2;
      Ints : UR_O2T_int_2;
      Floats : UR_O2T_floats_2;
END_STRUCT
END_TYPE

// ---- DUTs/UR_10 _O2T_Registers/UR_O2T_bits_2.TcDUT
TYPE UR_O2T_bits_2 :
   STRUCT
	B32:BIT;
	B33:BIT;
	B34:BIT;
	B35:BIT;
	B36:BIT;
	B37:BIT;
	B38:BIT;
	B39:BIT;
	B40:BIT;
	B41:BIT;
	B42:BIT;
	B43:BIT;
	B44:BIT;
	B45:BIT;
	B46:BIT;
	B47:BIT;
	B48:BIT;
	B49:BIT;
	B50:BIT;
	B51:BIT;
	B52:BIT;
	B53:BIT;
	B54:BIT;
	B55:BIT;
	B56:BIT;
	B57:BIT;
	B58:BIT;
	B59:BIT;
	B60:BIT;
	B61:BIT;
	B62:BIT;
	B63:BIT;
   END_STRUCT
END_TYPE

// ---- DUTs/UR_10 _O2T_Registers/UR_O2T_floats_2.TcDUT
TYPE UR_O2T_floats_2 :
STRUCT
FLOAT12:ARRAY[0..3] OF BYTE;
FLOAT13:ARRAY[0..3] OF BYTE;
FLOAT14:ARRAY[0..3] OF BYTE;
FLOAT15:ARRAY[0..3] OF BYTE;
FLOAT16:ARRAY[0..3] OF BYTE;
FLOAT17:ARRAY[0..3] OF BYTE;
FLOAT18:ARRAY[0..3] OF BYTE;
FLOAT19:ARRAY[0..3] OF BYTE;
FLOAT20:ARRAY[0..3] OF BYTE;
FLOAT21:ARRAY[0..3] OF BYTE;
FLOAT22:ARRAY[0..3] OF BYTE;
FLOAT23:ARRAY[0..3] OF BYTE;
END_STRUCT
END_TYPE

// ---- DUTs/UR_10 _O2T_Registers/UR_O2T_int_2.TcDUT
TYPE UR_O2T_int_2 :
STRUCT
INT12:ARRAY[0..3] OF BYTE;
INT13:ARRAY[0..3] OF BYTE;
INT14:ARRAY[0..3] OF BYTE;
INT15:ARRAY[0..3] OF BYTE;
INT16:ARRAY[0..3] OF BYTE;
INT17:ARRAY[0..3] OF BYTE;
INT18:ARRAY[0..3] OF BYTE;
INT19:ARRAY[0..3] OF BYTE;
INT20:ARRAY[0..3] OF BYTE;
INT21:ARRAY[0..3] OF BYTE;
INT22:ARRAY[0..3] OF BYTE;
INT23:ARRAY[0..3] OF BYTE;
END_STRUCT
END_TYPE

// ---- DUTs/UR_3_T2O_Joints/UR_3_T2O_Joints.TcDUT
TYPE UR_3_T2O_Joints :
STRUCT
FLOAT0:ARRAY[0..3] OF BYTE;
FLOAT1:ARRAY[0..3] OF BYTE;
FLOAT2:ARRAY[0..3] OF BYTE;
FLOAT3:ARRAY[0..3] OF BYTE;
FLOAT4:ARRAY[0..3] OF BYTE;
FLOAT5:ARRAY[0..3] OF BYTE;
END_STRUCT
END_TYPE

// ---- DUTs/UR_4_T2O_TCP/UR_4_T2O_TCP.TcDUT
TYPE UR_4_T2O_TCP :
STRUCT
FLOAT0:ARRAY[0..3] OF BYTE;
FLOAT1:ARRAY[0..3] OF BYTE;
FLOAT2:ARRAY[0..3] OF BYTE;
FLOAT3:ARRAY[0..3] OF BYTE;
FLOAT4:ARRAY[0..3] OF BYTE;
FLOAT5:ARRAY[0..3] OF BYTE;
FLOAT6:ARRAY[0..3] OF BYTE;
FLOAT7:ARRAY[0..3] OF BYTE;
FLOAT8:ARRAY[0..3] OF BYTE;
FLOAT9:ARRAY[0..3] OF BYTE;
FLOAT10:ARRAY[0..3] OF BYTE;
FLOAT11:ARRAY[0..3] OF BYTE;
FLOAT12:ARRAY[0..3] OF BYTE;
FLOAT13:ARRAY[0..3] OF BYTE;
FLOAT14:ARRAY[0..3] OF BYTE;
FLOAT15:ARRAY[0..3] OF BYTE;
FLOAT16:ARRAY[0..3] OF BYTE;
FLOAT17:ARRAY[0..3] OF BYTE;
FLOAT18:ARRAY[0..3] OF BYTE;
END_STRUCT
END_TYPE

// ---- DUTs/UR_5_T2O_BitRegisters/UR_5_T2O_BitRegisters.TcDUT
TYPE UR_5_T2O_BitRegisters :
STRUCT
	B0:BIT;
	B1:BIT;
	B2:BIT;
	B3:BIT;
	B4:BIT;
	B5:BIT;
	B6:BIT;
	B7:BIT;
	B8:BIT;
	B9:BIT;
	B10:BIT;
	B11:BIT;
	B12:BIT;
	B13:BIT;
	B14:BIT;
	B15:BIT;
	B16:BIT;
	B17:BIT;
	B18:BIT;
	B19:BIT;
	B20:BIT;
	B21:BIT;
	B22:BIT;
	B23:BIT;
	B24:BIT;
	B25:BIT;
	B26:BIT;
	B27:BIT;
	B28:BIT;
	B29:BIT;
	B30:BIT;
	B31:BIT;
	B32:BIT;
	B33:BIT;
	B34:BIT;
	B35:BIT;
	B36:BIT;
	B37:BIT;
	B38:BIT;
	B39:BIT;
	B40:BIT;
	B41:BIT;
	B42:BIT;
	B43:BIT;
	B44:BIT;
	B45:BIT;
	B46:BIT;
	B47:BIT;
	B48:BIT;
	B49:BIT;
	B50:BIT;
	B51:BIT;
	B52:BIT;
	B53:BIT;
	B54:BIT;
	B55:BIT;
	B56:BIT;
	B57:BIT;
	B58:BIT;
	B59:BIT;
	B60:BIT;
	B61:BIT;
	B62:BIT;
	B63:BIT;

END_STRUCT
END_TYPE

